LIN {X 0,Y 467.553,Z 325.87,A -85,B 0,C 180,E1 -7518.727,E2 -7518.727} C_VEL
LIN {X 0,Y 467.539,Z 325.868,A -85,B 0,C 180,E1 -7521.952,E2 -7521.952} C_VEL
LIN {X 0,Y 467.553,Z 325.867,A -85,B 0,C 180,E1 -7525.166,E2 -7525.166} C_VEL
LIN {X 0,Y 467.55,Z 325.866,A -85,B 0,C 180,E1 -7528.257,E2 -7528.257} C_VEL
LIN {X 0,Y 467.53,Z 325.867,A -85,B 0,C 180,E1 -7531.247,E2 -7531.247} C_VEL
LIN {X 0,Y 467.581,Z 325.868,A -85,B 0,C 180,E1 -7534.401,E2 -7534.401} C_VEL
LIN {X 0,Y 467.572,Z 325.861,A -85,B 0,C 180,E1 -7536.995,E2 -7536.995} C_VEL
LIN {X 0,Y 467.614,Z 325.847,A -85,B 0,C 180,E1 -7539.776,E2 -7539.776} C_VEL
LIN {X 0,Y 467.566,Z 325.869,A -85,B 0,C 180,E1 -7542.505,E2 -7542.505} C_VEL
LIN {X 0,Y 467.595,Z 325.86,A -85,B 0,C 180,E1 -7545.196,E2 -7545.196} C_VEL
LIN {X 0,Y 467.661,Z 325.849,A -85,B 0,C 180,E1 -7547.854,E2 -7547.854} C_VEL
LIN {X 0,Y 467.67,Z 325.846,A -85,B 0,C 180,E1 -7551.357,E2 -7551.357} C_VEL
LIN {X 0,Y 467.709,Z 325.851,A -85,B 0,C 180,E1 -7553.962,E2 -7553.962} C_VEL
LIN {X 0,Y 467.852,Z 325.827,A -85,B 0,C 180,E1 -7557.417,E2 -7557.417} C_VEL
LIN {X 0,Y 467.853,Z 325.834,A -85,B 0,C 180,E1 -7560,E2 -7560} C_VEL
LIN {X 0,Y 467.818,Z 325.834,A -85,B 0,C 180,E1 -7562.583,E2 -7562.583} C_VEL
LIN {X 0,Y 467.715,Z 325.85,A -85,B 0,C 180,E1 -7566.038,E2 -7566.038} C_VEL
LIN {X 0,Y 467.667,Z 325.852,A -85,B 0,C 180,E1 -7568.643,E2 -7568.643} C_VEL
LIN {X 0,Y 467.66,Z 325.857,A -85,B 0,C 180,E1 -7572.145,E2 -7572.145} C_VEL
LIN {X 0,Y 467.642,Z 325.858,A -85,B 0,C 180,E1 -7575.695,E2 -7575.695} C_VEL
LIN {X 0,Y 467.624,Z 325.857,A -85,B 0,C 180,E1 -7579.308,E2 -7579.308} C_VEL
LIN {X 0,Y 467.538,Z 325.872,A -85,B 0,C 180,E1 -7582.074,E2 -7582.074} C_VEL
LIN {X 0,Y 467.587,Z 325.861,A -85,B 0,C 180,E1 -7584.888,E2 -7584.888} C_VEL
LIN {X 0,Y 467.604,Z 325.867,A -85,B 0,C 180,E1 -7587.77,E2 -7587.77} C_VEL
LIN {X 0,Y 467.571,Z 325.866,A -85,B 0,C 180,E1 -7591.045,E2 -7591.045} C_VEL
LIN {X 0,Y 467.591,Z 325.864,A -85,B 0,C 180,E1 -7594.242,E2 -7594.242} C_VEL
LIN {X 0,Y 467.55,Z 325.87,A -85,B 0,C 180,E1 -7597.186,E2 -7597.186} C_VEL
LIN {X 0,Y 467.579,Z 325.864,A -85,B 0,C 180,E1 -7600.264,E2 -7600.264} C_VEL
LIN {X 0,Y 467.588,Z 325.863,A -85,B 0,C 180,E1 -7602.567,E2 -7602.567} C_VEL
LIN {X 0,Y 467.567,Z 325.867,A -85,B 0,C 180,E1 -7605.052,E2 -7605.052} C_VEL
LIN {X 0,Y 467.59,Z 325.868,A -85,B 0,C 180,E1 -7607.44,E2 -7607.44} C_VEL
LIN {X 0,Y 467.584,Z 325.865,A -85,B 0,C 180,E1 -7610.855,E2 -7610.855} C_VEL
LIN {X 0,Y 467.564,Z 325.869,A -85,B 0,C 180,E1 -7614.26,E2 -7614.26} C_VEL
LIN {X 0,Y 467.583,Z 325.87,A -85,B 0,C 180,E1 -7617.321,E2 -7617.321} C_VEL
LIN {X 0,Y 467.572,Z 325.868,A -85,B 0,C 180,E1 -7620.667,E2 -7620.667} C_VEL
LIN {X 0,Y 467.636,Z 325.967,A -85,B 0,C 180,E1 -7622.232,E2 -7622.232} C_VEL
LIN {X 0,Y 470.731,Z 340.487,A -85,B 0,C 180,E1 -7624.817,E2 -7624.817} C_VEL
LIN {X 0,Y 470.565,Z 347.239,A -85,B 0,C 180,E1 -7625.916,E2 -7625.916} C_VEL
LIN {X 0,Y 469.719,Z 364.781,A -85,B 0,C 180,E1 -7628.726,E2 -7628.726} C_VEL
LIN {X 0,Y 469.507,Z 369.211,A -85,B 0,C 180,E1 -7629.429,E2 -7629.429} C_VEL
LIN {X 0,Y 473.272,Z 391.149,A -85,B 0,C 180,E1 -7629.938,E2 -7629.938} C_VEL
LIN {X 0,Y 472.122,Z 507.018,A -85,B 0,C 180,E1 -7631.727,E2 -7631.727} C_VEL
LIN {X 0,Y 471.734,Z 521.803,A -85,B 0,C 180,E1 -7632.133,E2 -7632.133} C_VEL
LIN {X 0,Y 471.163,Z 535.874,A -85,B 0,C 180,E1 -7632.7,E2 -7632.7} C_VEL
LIN {X 0,Y 470.582,Z 549.218,A -85,B 0,C 180,E1 -7633.423,E2 -7633.423} C_VEL
LIN {X 0,Y 469.899,Z 561.559,A -85,B 0,C 180,E1 -7634.271,E2 -7634.271} C_VEL
LIN {X 0,Y 469.195,Z 573.089,A -85,B 0,C 180,E1 -7635.248,E2 -7635.248} C_VEL
LIN {X 0,Y 468.589,Z 583.675,A -85,B 0,C 180,E1 -7636.336,E2 -7636.336} C_VEL
LIN {X 0,Y 468.153,Z 593.303,A -85,B 0,C 180,E1 -7637.528,E2 -7637.528} C_VEL
LIN {X 0,Y 467.606,Z 602.867,A -85,B 0,C 180,E1 -7638.952,E2 -7638.952} C_VEL
LIN {X 0,Y 467.214,Z 611.173,A -85,B 0,C 180,E1 -7640.476,E2 -7640.476} C_VEL
LIN {X 0,Y 466.951,Z 616.974,A -85,B 0,C 180,E1 -7641.779,E2 -7641.779} C_VEL
LIN {X 0,Y 466.824,Z 621.734,A -85,B 0,C 180,E1 -7643.083,E2 -7643.083} C_VEL
LIN {X 0,Y 466.731,Z 626.661,A -85,B 0,C 180,E1 -7644.816,E2 -7644.816} C_VEL
LIN {X 0,Y 466.679,Z 630.085,A -85,B 0,C 180,E1 -7646.547,E2 -7646.547} C_VEL
LIN {X 0,Y 466.604,Z 632.11,A -85,B 0,C 180,E1 -7648.274,E2 -7648.274} C_VEL
LIN {X 0,Y 466.597,Z 632.785,A -85,B 0,C 180,E1 -7650,E2 -7650} C_VEL
LIN {X 0,Y 466.604,Z 632.119,A -85,B 0,C 180,E1 -7651.726,E2 -7651.726} C_VEL
LIN {X 0,Y 466.679,Z 630.105,A -85,B 0,C 180,E1 -7653.454,E2 -7653.454} C_VEL
LIN {X 0,Y 466.731,Z 626.693,A -85,B 0,C 180,E1 -7655.184,E2 -7655.184} C_VEL
LIN {X 0,Y 466.821,Z 621.783,A -85,B 0,C 180,E1 -7656.918,E2 -7656.918} C_VEL
LIN {X 0,Y 467.036,Z 615.238,A -85,B 0,C 180,E1 -7658.655,E2 -7658.655} C_VEL
LIN {X 0,Y 467.311,Z 607.962,A -85,B 0,C 180,E1 -7660.178,E2 -7660.178} C_VEL
LIN {X 0,Y 467.866,Z 598.973,A -85,B 0,C 180,E1 -7661.7,E2 -7661.7} C_VEL
LIN {X 0,Y 468.352,Z 589.547,A -85,B 0,C 180,E1 -7663.008,E2 -7663.008} C_VEL
LIN {X 0,Y 468.94,Z 579.125,A -85,B 0,C 180,E1 -7664.206,E2 -7664.206} C_VEL
LIN {X 0,Y 469.628,Z 567.65,A -85,B 0,C 180,E1 -7665.293,E2 -7665.293} C_VEL
LIN {X 0,Y 470.388,Z 554.947,A -85,B 0,C 180,E1 -7666.269,E2 -7666.269} C_VEL
LIN {X 0,Y 471.034,Z 542.365,A -85,B 0,C 180,E1 -7667.039,E2 -7667.039} C_VEL
LIN {X 0,Y 471.651,Z 528.534,A -85,B 0,C 180,E1 -7667.691,E2 -7667.691} C_VEL
LIN {X 0,Y 472.117,Z 514.909,A -85,B 0,C 180,E1 -7668.155,E2 -7668.155} C_VEL
LIN {X 0,Y 472.451,Z 501.171,A -85,B 0,C 180,E1 -7668.456,E2 -7668.456} C_VEL
LIN {X 0,Y 473.513,Z 390.833,A -85,B 0,C 180,E1 -7670.162,E2 -7670.162} C_VEL
LIN {X 0,Y 470.004,Z 371.054,A -85,B 0,C 180,E1 -7670.646,E2 -7670.646} C_VEL
LIN {X 0,Y 469.663,Z 369.039,A -85,B 0,C 180,E1 -7670.714,E2 -7670.714} C_VEL
LIN {X 0,Y 470.649,Z 350.152,A -85,B 0,C 180,E1 -7673.777,E2 -7673.777} C_VEL
LIN {X 0,Y 471.053,Z 341.727,A -85,B 0,C 180,E1 -7675.164,E2 -7675.164} C_VEL
LIN {X 0,Y 468.146,Z 328.134,A -85,B 0,C 180,E1 -7677.658,E2 -7677.658} C_VEL
LIN {X 0,Y 467.612,Z 325.864,A -85,B 0,C 180,E1 -7678.135,E2 -7678.135} C_VEL
LIN {X 0,Y 467.584,Z 325.863,A -85,B 0,C 180,E1 -7681.74,E2 -7681.74} C_VEL
LIN {X 0,Y 467.566,Z 325.87,A -85,B 0,C 180,E1 -7684.833,E2 -7684.833} C_VEL
LIN {X 0,Y 467.567,Z 325.868,A -85,B 0,C 180,E1 -7688.045,E2 -7688.045} C_VEL
LIN {X 0,Y 467.58,Z 325.863,A -85,B 0,C 180,E1 -7691.277,E2 -7691.277} C_VEL
LIN {X 0,Y 467.551,Z 325.866,A -85,B 0,C 180,E1 -7693.821,E2 -7693.821} C_VEL
LIN {X 0,Y 467.556,Z 325.869,A -85,B 0,C 180,E1 -7696.256,E2 -7696.256} C_VEL
LIN {X 0,Y 467.58,Z 325.866,A -85,B 0,C 180,E1 -7698.723,E2 -7698.723} C_VEL
LIN {X 0,Y 467.565,Z 325.866,A -85,B 0,C 180,E1 -7701.956,E2 -7701.956} C_VEL
LIN {X 0,Y 467.565,Z 325.865,A -85,B 0,C 180,E1 -7705.168,E2 -7705.168} C_VEL
LIN {X 0,Y 467.586,Z 325.868,A -85,B 0,C 180,E1 -7708.26,E2 -7708.26} C_VEL
LIN {X 0,Y 467.558,Z 325.865,A -85,B 0,C 180,E1 -7711.249,E2 -7711.249} C_VEL
LIN {X 0,Y 467.587,Z 325.864,A -85,B 0,C 180,E1 -7714.159,E2 -7714.159} C_VEL
LIN {X 0,Y 467.579,Z 325.861,A -85,B 0,C 180,E1 -7716.996,E2 -7716.996} C_VEL
LIN {X 0,Y 467.626,Z 325.859,A -85,B 0,C 180,E1 -7719.777,E2 -7719.777} C_VEL
LIN {X 0,Y 467.599,Z 325.861,A -85,B 0,C 180,E1 -7722.507,E2 -7722.507} C_VEL
LIN {X 0,Y 467.609,Z 325.859,A -85,B 0,C 180,E1 -7725.197,E2 -7725.197} C_VEL
LIN {X 0,Y 467.66,Z 325.853,A -85,B 0,C 180,E1 -7727.855,E2 -7727.855} C_VEL
LIN {X 0,Y 467.667,Z 325.85,A -85,B 0,C 180,E1 -7731.357,E2 -7731.357} C_VEL
LIN {X 0,Y 467.715,Z 325.853,A -85,B 0,C 180,E1 -7733.962,E2 -7733.962} C_VEL
LIN {X 0,Y 467.818,Z 325.829,A -85,B 0,C 180,E1 -7737.417,E2 -7737.417} C_VEL
LIN {X 0,Y 467.853,Z 325.833,A -85,B 0,C 180,E1 -7740,E2 -7740} C_VEL
LIN {X 0,Y 467.852,Z 325.827,A -85,B 0,C 180,E1 -7742.583,E2 -7742.583} C_VEL
LIN {X 0,Y 467.705,Z 325.846,A -85,B 0,C 180,E1 -7746.038,E2 -7746.038} C_VEL
LIN {X 0,Y 467.662,Z 325.852,A -85,B 0,C 180,E1 -7748.643,E2 -7748.643} C_VEL
LIN {X 0,Y 467.661,Z 325.853,A -85,B 0,C 180,E1 -7752.146,E2 -7752.146} C_VEL
LIN {X 0,Y 467.616,Z 325.86,A -85,B 0,C 180,E1 -7755.696,E2 -7755.696} C_VEL
LIN {X 0,Y 467.581,Z 325.862,A -85,B 0,C 180,E1 -7758.75,E2 -7758.75} C_VEL
LIN {X 0,Y 467.562,Z 325.864,A -85,B 0,C 180,E1 -7761.261,E2 -7761.261} C_VEL
LIN {X 0,Y 467.558,Z 325.865,A -85,B 0,C 180,E1 -7763.944,E2 -7763.944} C_VEL
LIN {X 0,Y 467.538,Z 325.868,A -85,B 0,C 180,E1 -7766.806,E2 -7766.806} C_VEL
LIN {X 0,Y 467.513,Z 325.861,A -85,B 0,C 180,E1 -7769.741,E2 -7769.741} C_VEL
LIN {X 0,Y 467.574,Z 325.862,A -85,B 0,C 180,E1 -7772.76,E2 -7772.76} C_VEL
LIN {X 0,Y 467.545,Z 325.859,A -85,B 0,C 180,E1 -7775.891,E2 -7775.891} C_VEL
LIN {X 0,Y 467.531,Z 325.873,A -85,B 0,C 180,E1 -7779.15,E2 -7779.15} C_VEL
LIN {X 0,Y 467.553,Z 325.873,A -85,B 0,C 180,E1 -7781.406,E2 -7781.406} C_VEL
LIN {X 0,Y 467.565,Z 325.869,A -85,B 0,C 180,E1 -7785.052,E2 -7785.052} C_VEL
LIN {X 0,Y 467.553,Z 325.87,A -85,B 0,C 180,E1 -7788.727,E2 -7788.727} C_VEL
LIN {X 0,Y 467.536,Z 325.872,A -85,B 0,C 180,E1 -7791.952,E2 -7791.952} C_VEL
LIN {X 0,Y 467.544,Z 325.874,A -85,B 0,C 180,E1 -7795.165,E2 -7795.165} C_VEL
LIN {X 0,Y 467.546,Z 325.868,A -85,B 0,C 180,E1 -7798.257,E2 -7798.257} C_VEL
LIN {X 0,Y 467.574,Z 326.065,A -85,B 0,C 180,E1 -7800.51,E2 -7800.51} C_VEL
LIN {X 0,Y 469.898,Z 337.319,A -85,B 0,C 180,E1 -7802.859,E2 -7802.859} C_VEL
LIN {X 0,Y 469.985,Z 342.162,A -85,B 0,C 180,E1 -7803.796,E2 -7803.796} C_VEL
LIN {X 0,Y 469.828,Z 345.296,A -85,B 0,C 180,E1 -7804.37,E2 -7804.37} C_VEL
LIN {X 0,Y 473.739,Z 362.985,A -85,B 0,C 180,E1 -7804.845,E2 -7804.845} C_VEL
LIN {X 0,Y 473.314,Z 405.55,A -85,B 0,C 180,E1 -7805.504,E2 -7805.504} C_VEL
LIN {X 0,Y 472.705,Z 411.397,A -85,B 0,C 180,E1 -7805.569,E2 -7805.569} C_VEL
LIN {X 0,Y 467.064,Z 430.434,A -85,B 0,C 180,E1 -7805.612,E2 -7805.612} C_VEL
LIN {X 0,Y 466.356,Z 436.288,A -85,B 0,C 180,E1 -7805.674,E2 -7805.674} C_VEL
LIN {X 0,Y 465.947,Z 481.822,A -85,B 0,C 180,E1 -7806.411,E2 -7806.411} C_VEL
LIN {X 0,Y 465.524,Z 495.912,A -85,B 0,C 180,E1 -7806.8,E2 -7806.8} C_VEL
LIN {X 0,Y 464.986,Z 508.239,A -85,B 0,C 180,E1 -7807.288,E2 -7807.288} C_VEL
LIN {X 0,Y 464.373,Z 521.643,A -85,B 0,C 180,E1 -7808.002,E2 -7808.002} C_VEL
LIN {X 0,Y 463.638,Z 534.729,A -85,B 0,C 180,E1 -7808.899,E2 -7808.899} C_VEL
LIN {X 0,Y 462.972,Z 545.605,A -85,B 0,C 180,E1 -7809.82,E2 -7809.82} C_VEL
LIN {X 0,Y 462.286,Z 556.356,A -85,B 0,C 180,E1 -7810.922,E2 -7810.922} C_VEL
LIN {X 0,Y 461.558,Z 567.169,A -85,B 0,C 180,E1 -7812.27,E2 -7812.27} C_VEL
LIN {X 0,Y 461.008,Z 576.208,A -85,B 0,C 180,E1 -7813.643,E2 -7813.643} C_VEL
LIN {X 0,Y 460.571,Z 583.422,A -85,B 0,C 180,E1 -7814.965,E2 -7814.965} C_VEL
LIN {X 0,Y 460.181,Z 589.526,A -85,B 0,C 180,E1 -7816.307,E2 -7816.307} C_VEL
LIN {X 0,Y 459.834,Z 595.712,A -85,B 0,C 180,E1 -7818.006,E2 -7818.006} C_VEL
LIN {X 0,Y 459.725,Z 599.724,A -85,B 0,C 180,E1 -7819.429,E2 -7819.429} C_VEL
LIN {X 0,Y 459.57,Z 603.358,A -85,B 0,C 180,E1 -7821.203,E2 -7821.203} C_VEL
LIN {X 0,Y 459.576,Z 605.577,A -85,B 0,C 180,E1 -7822.973,E2 -7822.973} C_VEL
LIN {X 0,Y 459.558,Z 606.452,A -85,B 0,C 180,E1 -7824.735,E2 -7824.735} C_VEL
LIN {X 0,Y 459.563,Z 606.007,A -85,B 0,C 180,E1 -7826.493,E2 -7826.493} C_VEL
LIN {X 0,Y 459.572,Z 604.245,A -85,B 0,C 180,E1 -7828.247,E2 -7828.247} C_VEL
LIN {X 0,Y 459.571,Z 601.136,A -85,B 0,C 180,E1 -7830,E2 -7830} C_VEL
LIN {X 0,Y 459.707,Z 596.563,A -85,B 0,C 180,E1 -7831.752,E2 -7831.752} C_VEL
LIN {X 0,Y 460.099,Z 590.362,A -85,B 0,C 180,E1 -7833.503,E2 -7833.503} C_VEL
LIN {X 0,Y 460.54,Z 583.469,A -85,B 0,C 180,E1 -7835.034,E2 -7835.034} C_VEL
LIN {X 0,Y 461.001,Z 574.951,A -85,B 0,C 180,E1 -7836.565,E2 -7836.565} C_VEL
LIN {X 0,Y 461.415,Z 567.702,A -85,B 0,C 180,E1 -7837.654,E2 -7837.654} C_VEL
LIN {X 0,Y 461.983,Z 559.151,A -85,B 0,C 180,E1 -7838.75,E2 -7838.75} C_VEL
LIN {X 0,Y 462.709,Z 547.862,A -85,B 0,C 180,E1 -7839.949,E2 -7839.949} C_VEL
LIN {X 0,Y 463.353,Z 536.647,A -85,B 0,C 180,E1 -7840.929,E2 -7840.929} C_VEL
LIN {X 0,Y 464.007,Z 524.401,A -85,B 0,C 180,E1 -7841.799,E2 -7841.799} C_VEL
LIN {X 0,Y 464.565,Z 510.773,A -85,B 0,C 180,E1 -7842.56,E2 -7842.56} C_VEL
LIN {X 0,Y 465.159,Z 497.073,A -85,B 0,C 180,E1 -7843.127,E2 -7843.127} C_VEL
LIN {X 0,Y 465.47,Z 482.92,A -85,B 0,C 180,E1 -7843.535,E2 -7843.535} C_VEL
LIN {X 0,Y 465.999,Z 437.32,A -85,B 0,C 180,E1 -7844.269,E2 -7844.269} C_VEL
LIN {X 0,Y 466.607,Z 363.158,A -85,B 0,C 180,E1 -7845.427,E2 -7845.427} C_VEL
LIN {X 0,Y 462.751,Z 345.257,A -85,B 0,C 180,E1 -7845.893,E2 -7845.893} C_VEL
LIN {X 0,Y 462.849,Z 338.115,A -85,B 0,C 180,E1 -7847.252,E2 -7847.252} C_VEL
LIN {X 0,Y 460.57,Z 326.743,A -85,B 0,C 180,E1 -7849.616,E2 -7849.616} C_VEL
LIN {X 0,Y 460.499,Z 326.75,A -85,B 0,C 180,E1 -7852.429,E2 -7852.429} C_VEL
LIN {X 0,Y 460.524,Z 326.745,A -85,B 0,C 180,E1 -7855.789,E2 -7855.789} C_VEL
LIN {X 0,Y 460.499,Z 326.748,A -85,B 0,C 180,E1 -7858.237,E2 -7858.237} C_VEL
LIN {X 0,Y 460.499,Z 326.748,A -85,B 0,C 180,E1 -7861.277,E2 -7861.277} C_VEL
LIN {X 0,Y 460.512,Z 326.748,A -85,B 0,C 180,E1 -7864.501,E2 -7864.501} C_VEL
LIN {X 0,Y 460.481,Z 326.747,A -85,B 0,C 180,E1 -7867.625,E2 -7867.625} C_VEL
LIN {X 0,Y 460.502,Z 326.747,A -85,B 0,C 180,E1 -7871.015,E2 -7871.015} C_VEL
LIN {X 0,Y 460.513,Z 326.748,A -85,B 0,C 180,E1 -7874.589,E2 -7874.589} C_VEL
LIN {X 0,Y 460.473,Z 326.747,A -85,B 0,C 180,E1 -7877.812,E2 -7877.812} C_VEL
LIN {X 0,Y 460.477,Z 326.749,A -85,B 0,C 180,E1 -7880.131,E2 -7880.131} C_VEL
LIN {X 0,Y 460.461,Z 326.747,A -85,B 0,C 180,E1 -7883.469,E2 -7883.469} C_VEL
LIN {X 0,Y 460.518,Z 326.743,A -85,B 0,C 180,E1 -7886.674,E2 -7886.674} C_VEL
LIN {X 0,Y 460.482,Z 326.747,A -85,B 0,C 180,E1 -7889.757,E2 -7889.757} C_VEL
LIN {X 0,Y 460.493,Z 326.746,A -85,B 0,C 180,E1 -7892.751,E2 -7892.751} C_VEL
LIN {X 0,Y 460.52,Z 326.742,A -85,B 0,C 180,E1 -7895.666,E2 -7895.666} C_VEL
LIN {X 0,Y 460.522,Z 326.734,A -85,B 0,C 180,E1 -7898.579,E2 -7898.579} C_VEL
LIN {X 0,Y 460.585,Z 326.727,A -85,B 0,C 180,E1 -7901.31,E2 -7901.31} C_VEL
LIN {X 0,Y 460.552,Z 326.738,A -85,B 0,C 180,E1 -7904.964,E2 -7904.964} C_VEL
LIN {X 0,Y 460.613,Z 326.717,A -85,B 0,C 180,E1 -7908.559,E2 -7908.559} C_VEL
LIN {X 0,Y 460.621,Z 326.724,A -85,B 0,C 180,E1 -7911.223,E2 -7911.223} C_VEL
LIN {X 0,Y 460.675,Z 326.726,A -85,B 0,C 180,E1 -7913.869,E2 -7913.869} C_VEL
LIN {X 0,Y 460.792,Z 326.707,A -85,B 0,C 180,E1 -7917.377,E2 -7917.377} C_VEL
LIN {X 0,Y 460.823,Z 326.71,A -85,B 0,C 180,E1 -7920,E2 -7920} C_VEL
LIN {X 0,Y 460.762,Z 326.713,A -85,B 0,C 180,E1 -7922.622,E2 -7922.622} C_VEL
LIN {X 0,Y 460.679,Z 326.727,A -85,B 0,C 180,E1 -7926.13,E2 -7926.13} C_VEL
LIN {X 0,Y 460.618,Z 326.729,A -85,B 0,C 180,E1 -7928.776,E2 -7928.776} C_VEL
LIN {X 0,Y 460.617,Z 326.731,A -85,B 0,C 180,E1 -7932.445,E2 -7932.445} C_VEL
LIN {X 0,Y 460.604,Z 326.738,A -85,B 0,C 180,E1 -7935.997,E2 -7935.997} C_VEL
LIN {X 0,Y 460.571,Z 326.739,A -85,B 0,C 180,E1 -7939.615,E2 -7939.615} C_VEL
LIN {X 0,Y 460.514,Z 326.743,A -85,B 0,C 180,E1 -7942.428,E2 -7942.428} C_VEL
LIN {X 0,Y 460.548,Z 326.744,A -85,B 0,C 180,E1 -7945.796,E2 -7945.796} C_VEL
LIN {X 0,Y 460.538,Z 326.741,A -85,B 0,C 180,E1 -7948.234,E2 -7948.234} C_VEL
LIN {X 0,Y 460.523,Z 326.746,A -85,B 0,C 180,E1 -7951.283,E2 -7951.283} C_VEL
LIN {X 0,Y 460.534,Z 326.742,A -85,B 0,C 180,E1 -7954.505,E2 -7954.505} C_VEL
LIN {X 0,Y 460.529,Z 326.749,A -85,B 0,C 180,E1 -7957.62,E2 -7957.62} C_VEL
LIN {X 0,Y 460.544,Z 326.741,A -85,B 0,C 180,E1 -7960.269,E2 -7960.269} C_VEL
LIN {X 0,Y 460.501,Z 326.751,A -85,B 0,C 180,E1 -7963.375,E2 -7963.375} C_VEL
LIN {X 0,Y 460.5,Z 326.745,A -85,B 0,C 180,E1 -7966.624,E2 -7966.624} C_VEL
LIN {X 0,Y 460.543,Z 326.745,A -85,B 0,C 180,E1 -7969.73,E2 -7969.73} C_VEL
LIN {X 0,Y 460.528,Z 326.745,A -85,B 0,C 180,E1 -7972.519,E2 -7972.519} C_VEL
LIN {X 0,Y 460.55,Z 326.746,A -85,B 0,C 180,E1 -7975.624,E2 -7975.624} C_VEL
LIN {X 0,Y 460.538,Z 326.743,A -85,B 0,C 180,E1 -7978.744,E2 -7978.744} C_VEL
LIN {X 0,Y 460.593,Z 326.831,A -85,B 0,C 180,E1 -7981.979,E2 -7981.979} C_VEL
LIN {X 0,Y 463.754,Z 341.584,A -85,B 0,C 180,E1 -7984.652,E2 -7984.652} C_VEL
LIN {X 0,Y 463.763,Z 346.87,A -85,B 0,C 180,E1 -7985.533,E2 -7985.533} C_VEL
LIN {X 0,Y 462.75,Z 365.877,A -85,B 0,C 180,E1 -7988.623,E2 -7988.623} C_VEL
LIN {X 0,Y 462.598,Z 369.02,A -85,B 0,C 180,E1 -7989.131,E2 -7989.131} C_VEL
LIN {X 0,Y 466.544,Z 392.063,A -85,B 0,C 180,E1 -7989.673,E2 -7989.673} C_VEL
LIN {X 0,Y 465.333,Z 507.257,A -85,B 0,C 180,E1 -7991.48,E2 -7991.48} C_VEL
LIN {X 0,Y 464.919,Z 521.888,A -85,B 0,C 180,E1 -7991.89,E2 -7991.89} C_VEL
LIN {X 0,Y 464.342,Z 535.865,A -85,B 0,C 180,E1 -7992.464,E2 -7992.464} C_VEL
LIN {X 0,Y 463.733,Z 548.889,A -85,B 0,C 180,E1 -7993.18,E2 -7993.18} C_VEL
LIN {X 0,Y 463.03,Z 561.144,A -85,B 0,C 180,E1 -7994.032,E2 -7994.032} C_VEL
LIN {X 0,Y 462.289,Z 572.719,A -85,B 0,C 180,E1 -7995.022,E2 -7995.022} C_VEL
LIN {X 0,Y 461.632,Z 583.336,A -85,B 0,C 180,E1 -7996.126,E2 -7996.126} C_VEL
LIN {X 0,Y 461.123,Z 593.72,A -85,B 0,C 180,E1 -7997.434,E2 -7997.434} C_VEL
LIN {X 0,Y 460.601,Z 602.579,A -85,B 0,C 180,E1 -7998.782,E2 -7998.782} C_VEL
LIN {X 0,Y 460.142,Z 610.908,A -85,B 0,C 180,E1 -8000.328,E2 -8000.328} C_VEL
LIN {X 0,Y 459.896,Z 616.719,A -85,B 0,C 180,E1 -8001.652,E2 -8001.652} C_VEL
LIN {X 0,Y 459.733,Z 621.492,A -85,B 0,C 180,E1 -8002.975,E2 -8002.975} C_VEL
LIN {X 0,Y 459.644,Z 626.432,A -85,B 0,C 180,E1 -8004.736,E2 -8004.736} C_VEL
LIN {X 0,Y 459.574,Z 629.866,A -85,B 0,C 180,E1 -8006.493,E2 -8006.493} C_VEL
LIN {X 0,Y 459.517,Z 631.9,A -85,B 0,C 180,E1 -8008.247,E2 -8008.247} C_VEL
LIN {X 0,Y 459.528,Z 632.584,A -85,B 0,C 180,E1 -8010,E2 -8010} C_VEL
LIN {X 0,Y 459.517,Z 631.926,A -85,B 0,C 180,E1 -8011.753,E2 -8011.753} C_VEL
LIN {X 0,Y 459.574,Z 629.92,A -85,B 0,C 180,E1 -8013.507,E2 -8013.507} C_VEL
LIN {X 0,Y 459.645,Z 626.518,A -85,B 0,C 180,E1 -8015.264,E2 -8015.264} C_VEL
LIN {X 0,Y 459.731,Z 621.621,A -85,B 0,C 180,E1 -8017.025,E2 -8017.025} C_VEL
LIN {X 0,Y 459.969,Z 615.089,A -85,B 0,C 180,E1 -8018.789,E2 -8018.789} C_VEL
LIN {X 0,Y 460.28,Z 607.829,A -85,B 0,C 180,E1 -8020.336,E2 -8020.336} C_VEL
LIN {X 0,Y 460.856,Z 598.866,A -85,B 0,C 180,E1 -8021.881,E2 -8021.881} C_VEL
LIN {X 0,Y 461.374,Z 589.468,A -85,B 0,C 180,E1 -8023.208,E2 -8023.208} C_VEL
LIN {X 0,Y 462.008,Z 579.079,A -85,B 0,C 180,E1 -8024.424,E2 -8024.424} C_VEL
LIN {X 0,Y 462.766,Z 567.642,A -85,B 0,C 180,E1 -8025.526,E2 -8025.526} C_VEL
LIN {X 0,Y 463.561,Z 554.989,A -85,B 0,C 180,E1 -8026.515,E2 -8026.515} C_VEL
LIN {X 0,Y 464.308,Z 541.922,A -85,B 0,C 180,E1 -8027.326,E2 -8027.326} C_VEL
LIN {X 0,Y 464.905,Z 527.983,A -85,B 0,C 180,E1 -8027.99,E2 -8027.99} C_VEL
LIN {X 0,Y 465.475,Z 513.268,A -85,B 0,C 180,E1 -8028.486,E2 -8028.486} C_VEL
LIN {X 0,Y 465.787,Z 498.747,A -85,B 0,C 180,E1 -8028.787,E2 -8028.787} C_VEL
LIN {X 0,Y 466.906,Z 391.754,A -85,B 0,C 180,E1 -8030.462,E2 -8030.462} C_VEL
LIN {X 0,Y 463.435,Z 372.229,A -85,B 0,C 180,E1 -8030.951,E2 -8030.951} C_VEL
LIN {X 0,Y 462.798,Z 368.937,A -85,B 0,C 180,E1 -8031.04,E2 -8031.04} C_VEL
LIN {X 0,Y 463.768,Z 351.507,A -85,B 0,C 180,E1 -8033.915,E2 -8033.915} C_VEL
LIN {X 0,Y 464.155,Z 343.091,A -85,B 0,C 180,E1 -8035.325,E2 -8035.325} C_VEL
LIN {X 0,Y 461.437,Z 330.397,A -85,B 0,C 180,E1 -8037.694,E2 -8037.694} C_VEL
LIN {X 0,Y 460.575,Z 326.74,A -85,B 0,C 180,E1 -8038.418,E2 -8038.418} C_VEL
LIN {X 0,Y 460.523,Z 326.744,A -85,B 0,C 180,E1 -8041.283,E2 -8041.283} C_VEL
LIN {X 0,Y 460.533,Z 326.747,A -85,B 0,C 180,E1 -8044.506,E2 -8044.506} C_VEL
LIN {X 0,Y 460.503,Z 326.746,A -85,B 0,C 180,E1 -8047.623,E2 -8047.623} C_VEL
LIN {X 0,Y 460.541,Z 326.744,A -85,B 0,C 180,E1 -8050.269,E2 -8050.269} C_VEL
LIN {X 0,Y 460.498,Z 326.743,A -85,B 0,C 180,E1 -8053.376,E2 -8053.376} C_VEL
LIN {X 0,Y 460.501,Z 326.75,A -85,B 0,C 180,E1 -8056.625,E2 -8056.625} C_VEL
LIN {X 0,Y 460.544,Z 326.74,A -85,B 0,C 180,E1 -8059.731,E2 -8059.731} C_VEL
LIN {X 0,Y 460.499,Z 326.748,A -85,B 0,C 180,E1 -8062.525,E2 -8062.525} C_VEL
LIN {X 0,Y 460.548,Z 326.739,A -85,B 0,C 180,E1 -8065.624,E2 -8065.624} C_VEL
LIN {X 0,Y 460.54,Z 326.741,A -85,B 0,C 180,E1 -8068.745,E2 -8068.745} C_VEL
LIN {X 0,Y 460.553,Z 326.744,A -85,B 0,C 180,E1 -8072.262,E2 -8072.262} C_VEL
LIN {X 0,Y 460.543,Z 326.741,A -85,B 0,C 180,E1 -8074.705,E2 -8074.705} C_VEL
LIN {X 0,Y 460.514,Z 326.742,A -85,B 0,C 180,E1 -8077.572,E2 -8077.572} C_VEL
LIN {X 0,Y 460.571,Z 326.739,A -85,B 0,C 180,E1 -8080.385,E2 -8080.385} C_VEL
LIN {X 0,Y 460.608,Z 326.737,A -85,B 0,C 180,E1 -8084.059,E2 -8084.059} C_VEL
LIN {X 0,Y 460.613,Z 326.728,A -85,B 0,C 180,E1 -8087.666,E2 -8087.666} C_VEL
LIN {X 0,Y 460.619,Z 326.727,A -85,B 0,C 180,E1 -8091.224,E2 -8091.224} C_VEL
LIN {X 0,Y 460.679,Z 326.727,A -85,B 0,C 180,E1 -8093.87,E2 -8093.87} C_VEL
LIN {X 0,Y 460.762,Z 326.708,A -85,B 0,C 180,E1 -8097.378,E2 -8097.378} C_VEL
LIN {X 0,Y 460.823,Z 326.708,A -85,B 0,C 180,E1 -8100,E2 -8100} C_VEL
LIN {X 0,Y 460.792,Z 326.706,A -85,B 0,C 180,E1 -8102.623,E2 -8102.623} C_VEL
LIN {X 0,Y 460.671,Z 326.721,A -85,B 0,C 180,E1 -8106.131,E2 -8106.131} C_VEL
LIN {X 0,Y 460.614,Z 326.73,A -85,B 0,C 180,E1 -8108.777,E2 -8108.777} C_VEL
LIN {X 0,Y 460.614,Z 326.729,A -85,B 0,C 180,E1 -8112.334,E2 -8112.334} C_VEL
LIN {X 0,Y 460.561,Z 326.736,A -85,B 0,C 180,E1 -8115.978,E2 -8115.978} C_VEL
LIN {X 0,Y 460.539,Z 326.74,A -85,B 0,C 180,E1 -8118.888,E2 -8118.888} C_VEL
LIN {X 0,Y 460.513,Z 326.744,A -85,B 0,C 180,E1 -8121.486,E2 -8121.486} C_VEL
LIN {X 0,Y 460.521,Z 326.739,A -85,B 0,C 180,E1 -8124.334,E2 -8124.334} C_VEL
LIN {X 0,Y 460.493,Z 326.75,A -85,B 0,C 180,E1 -8127.249,E2 -8127.249} C_VEL
LIN {X 0,Y 460.481,Z 326.733,A -85,B 0,C 180,E1 -8130.243,E2 -8130.243} C_VEL
LIN {X 0,Y 460.519,Z 326.747,A -85,B 0,C 180,E1 -8133.326,E2 -8133.326} C_VEL
LIN {X 0,Y 460.46,Z 326.738,A -85,B 0,C 180,E1 -8136.531,E2 -8136.531} C_VEL
LIN {X 0,Y 460.477,Z 326.748,A -85,B 0,C 180,E1 -8139.869,E2 -8139.869} C_VEL
LIN {X 0,Y 460.46,Z 326.752,A -85,B 0,C 180,E1 -8142.893,E2 -8142.893} C_VEL
LIN {X 0,Y 460.507,Z 326.743,A -85,B 0,C 180,E1 -8145.832,E2 -8145.832} C_VEL
LIN {X 0,Y 460.502,Z 326.748,A -85,B 0,C 180,E1 -8148.985,E2 -8148.985} C_VEL
LIN {X 0,Y 460.481,Z 326.75,A -85,B 0,C 180,E1 -8152.375,E2 -8152.375} C_VEL
LIN {X 0,Y 460.526,Z 326.745,A -85,B 0,C 180,E1 -8155.622,E2 -8155.622} C_VEL
LIN {X 0,Y 460.508,Z 326.748,A -85,B 0,C 180,E1 -8158.742,E2 -8158.742} C_VEL
LIN {X 0,Y 460.489,Z 326.821,A -85,B 0,C 180,E1 -8160.194,E2 -8160.194} C_VEL
LIN {X 0,Y 462.943,Z 338.423,A -85,B 0,C 180,E1 -8162.662,E2 -8162.662} C_VEL
LIN {X 0,Y 463.135,Z 342.907,A -85,B 0,C 180,E1 -8163.55,E2 -8163.55} C_VEL
LIN {X 0,Y 463.039,Z 345.659,A -85,B 0,C 180,E1 -8164.033,E2 -8164.033} C_VEL
LIN {X 0,Y 467.072,Z 363.728,A -85,B 0,C 180,E1 -8164.532,E2 -8164.532} C_VEL
LIN {X 0,Y 466.356,Z 436.288,A -85,B 0,C 180,E1 -8165.674,E2 -8165.674} C_VEL
LIN {X 0,Y 465.687,Z 442.128,A -85,B 0,C 180,E1 -8165.737,E2 -8165.737} C_VEL
LIN {X 0,Y 460.198,Z 461.163,A -85,B 0,C 180,E1 -8165.788,E2 -8165.788} C_VEL
LIN {X 0,Y 459.468,Z 467.007,A -85,B 0,C 180,E1 -8165.849,E2 -8165.849} C_VEL
LIN {X 0,Y 459.186,Z 485.434,A -85,B 0,C 180,E1 -8166.191,E2 -8166.191} C_VEL
LIN {X 0,Y 458.667,Z 499.82,A -85,B 0,C 180,E1 -8166.638,E2 -8166.638} C_VEL
LIN {X 0,Y 458.115,Z 513.131,A -85,B 0,C 180,E1 -8167.233,E2 -8167.233} C_VEL
LIN {X 0,Y 457.405,Z 526.288,A -85,B 0,C 180,E1 -8168.005,E2 -8168.005} C_VEL
LIN {X 0,Y 456.64,Z 538.493,A -85,B 0,C 180,E1 -8168.915,E2 -8168.915} C_VEL
LIN {X 0,Y 455.901,Z 549.895,A -85,B 0,C 180,E1 -8169.964,E2 -8169.964} C_VEL
LIN {X 0,Y 455.165,Z 559.958,A -85,B 0,C 180,E1 -8171.08,E2 -8171.08} C_VEL
LIN {X 0,Y 454.435,Z 570.128,A -85,B 0,C 180,E1 -8172.448,E2 -8172.448} C_VEL
LIN {X 0,Y 453.902,Z 578.54,A -85,B 0,C 180,E1 -8173.817,E2 -8173.817} C_VEL
LIN {X 0,Y 453.346,Z 586.545,A -85,B 0,C 180,E1 -8175.409,E2 -8175.409} C_VEL
LIN {X 0,Y 452.989,Z 592.958,A -85,B 0,C 180,E1 -8176.999,E2 -8176.999} C_VEL
LIN {X 0,Y 452.69,Z 598.617,A -85,B 0,C 180,E1 -8178.81,E2 -8178.81} C_VEL
LIN {X 0,Y 452.524,Z 601.803,A -85,B 0,C 180,E1 -8180.163,E2 -8180.163} C_VEL
LIN {X 0,Y 452.477,Z 604.763,A -85,B 0,C 180,E1 -8181.964,E2 -8181.964} C_VEL
LIN {X 0,Y 452.518,Z 606.347,A -85,B 0,C 180,E1 -8183.759,E2 -8183.759} C_VEL
LIN {X 0,Y 452.435,Z 606.607,A -85,B 0,C 180,E1 -8185.545,E2 -8185.545} C_VEL
LIN {X 0,Y 452.516,Z 605.547,A -85,B 0,C 180,E1 -8187.329,E2 -8187.329} C_VEL
LIN {X 0,Y 452.466,Z 603.165,A -85,B 0,C 180,E1 -8189.11,E2 -8189.11} C_VEL
LIN {X 0,Y 452.55,Z 599.399,A -85,B 0,C 180,E1 -8190.89,E2 -8190.89} C_VEL
LIN {X 0,Y 452.83,Z 594.093,A -85,B 0,C 180,E1 -8192.669,E2 -8192.669} C_VEL
LIN {X 0,Y 453.226,Z 589.013,A -85,B 0,C 180,E1 -8194.001,E2 -8194.001} C_VEL
LIN {X 0,Y 453.644,Z 581.763,A -85,B 0,C 180,E1 -8195.556,E2 -8195.556} C_VEL
LIN {X 0,Y 454.202,Z 572.769,A -85,B 0,C 180,E1 -8197.111,E2 -8197.111} C_VEL
LIN {X 0,Y 454.591,Z 564.937,A -85,B 0,C 180,E1 -8198.243,E2 -8198.243} C_VEL
LIN {X 0,Y 455.428,Z 554.025,A -85,B 0,C 180,E1 -8199.549,E2 -8199.549} C_VEL
LIN {X 0,Y 456.101,Z 542.773,A -85,B 0,C 180,E1 -8200.656,E2 -8200.656} C_VEL
LIN {X 0,Y 456.838,Z 530.327,A -85,B 0,C 180,E1 -8201.649,E2 -8201.649} C_VEL
LIN {X 0,Y 457.482,Z 518.286,A -85,B 0,C 180,E1 -8202.42,E2 -8202.42} C_VEL
LIN {X 0,Y 458.086,Z 506.307,A -85,B 0,C 180,E1 -8203.023,E2 -8203.023} C_VEL
LIN {X 0,Y 458.513,Z 492.369,A -85,B 0,C 180,E1 -8203.546,E2 -8203.546} C_VEL
LIN {X 0,Y 458.789,Z 479.205,A -85,B 0,C 180,E1 -8203.877,E2 -8203.877} C_VEL
LIN {X 0,Y 459.926,Z 364.299,A -85,B 0,C 180,E1 -8205.699,E2 -8205.699} C_VEL
LIN {X 0,Y 455.878,Z 345.462,A -85,B 0,C 180,E1 -8206.197,E2 -8206.197} C_VEL
LIN {X 0,Y 456.044,Z 340.44,A -85,B 0,C 180,E1 -8207.161,E2 -8207.161} C_VEL
LIN {X 0,Y 453.511,Z 327.622,A -85,B 0,C 180,E1 -8209.854,E2 -8209.854} C_VEL
LIN {X 0,Y 453.467,Z 327.628,A -85,B 0,C 180,E1 -8212.797,E2 -8212.797} C_VEL
LIN {X 0,Y 453.469,Z 327.624,A -85,B 0,C 180,E1 -8215.985,E2 -8215.985} C_VEL
LIN {X 0,Y 453.451,Z 327.63,A -85,B 0,C 180,E1 -8218.716,E2 -8218.716} C_VEL
LIN {X 0,Y 453.437,Z 327.625,A -85,B 0,C 180,E1 -8221.802,E2 -8221.802} C_VEL
LIN {X 0,Y 453.469,Z 327.626,A -85,B 0,C 180,E1 -8224.99,E2 -8224.99} C_VEL
LIN {X 0,Y 453.44,Z 327.627,A -85,B 0,C 180,E1 -8228.314,E2 -8228.314} C_VEL
LIN {X 0,Y 453.467,Z 327.627,A -85,B 0,C 180,E1 -8230.612,E2 -8230.612} C_VEL
LIN {X 0,Y 453.483,Z 327.624,A -85,B 0,C 180,E1 -8234.528,E2 -8234.528} C_VEL
LIN {X 0,Y 453.433,Z 327.626,A -85,B 0,C 180,E1 -8238.072,E2 -8238.072} C_VEL
LIN {X 0,Y 453.426,Z 327.63,A -85,B 0,C 180,E1 -8240.804,E2 -8240.804} C_VEL
LIN {X 0,Y 453.444,Z 327.623,A -85,B 0,C 180,E1 -8243.916,E2 -8243.916} C_VEL
LIN {X 0,Y 453.483,Z 327.617,A -85,B 0,C 180,E1 -8246.813,E2 -8246.813} C_VEL
LIN {X 0,Y 453.45,Z 327.628,A -85,B 0,C 180,E1 -8250.266,E2 -8250.266} C_VEL
LIN {X 0,Y 453.444,Z 327.62,A -85,B 0,C 180,E1 -8253.29,E2 -8253.29} C_VEL
LIN {X 0,Y 453.495,Z 327.623,A -85,B 0,C 180,E1 -8256.238,E2 -8256.238} C_VEL
LIN {X 0,Y 453.477,Z 327.606,A -85,B 0,C 180,E1 -8259.117,E2 -8259.117} C_VEL
LIN {X 0,Y 453.487,Z 327.614,A -85,B 0,C 180,E1 -8261.943,E2 -8261.943} C_VEL
LIN {X 0,Y 453.522,Z 327.615,A -85,B 0,C 180,E1 -8264.725,E2 -8264.725} C_VEL
LIN {X 0,Y 453.562,Z 327.596,A -85,B 0,C 180,E1 -8268.379,E2 -8268.379} C_VEL
LIN {X 0,Y 453.587,Z 327.6,A -85,B 0,C 180,E1 -8271.086,E2 -8271.086} C_VEL
LIN {X 0,Y 453.642,Z 327.601,A -85,B 0,C 180,E1 -8273.774,E2 -8273.774} C_VEL
LIN {X 0,Y 453.736,Z 327.585,A -85,B 0,C 180,E1 -8277.336,E2 -8277.336} C_VEL
LIN {X 0,Y 453.792,Z 327.585,A -85,B 0,C 180,E1 -8280,E2 -8280} C_VEL
LIN {X 0,Y 453.709,Z 327.591,A -85,B 0,C 180,E1 -8282.663,E2 -8282.663} C_VEL
LIN {X 0,Y 453.646,Z 327.603,A -85,B 0,C 180,E1 -8286.226,E2 -8286.226} C_VEL
LIN {X 0,Y 453.585,Z 327.605,A -85,B 0,C 180,E1 -8288.913,E2 -8288.913} C_VEL
LIN {X 0,Y 453.567,Z 327.609,A -85,B 0,C 180,E1 -8292.529,E2 -8292.529} C_VEL
LIN {X 0,Y 453.547,Z 327.614,A -85,B 0,C 180,E1 -8296.196,E2 -8296.196} C_VEL
LIN {X 0,Y 453.519,Z 327.612,A -85,B 0,C 180,E1 -8299.039,E2 -8299.039} C_VEL
LIN {X 0,Y 453.479,Z 327.623,A -85,B 0,C 180,E1 -8301.836,E2 -8301.836} C_VEL
LIN {X 0,Y 453.502,Z 327.616,A -85,B 0,C 180,E1 -8304.735,E2 -8304.735} C_VEL
LIN {X 0,Y 453.52,Z 327.619,A -85,B 0,C 180,E1 -8307.956,E2 -8307.956} C_VEL
LIN {X 0,Y 453.468,Z 327.627,A -85,B 0,C 180,E1 -8311.525,E2 -8311.525} C_VEL
LIN {X 0,Y 453.49,Z 327.619,A -85,B 0,C 180,E1 -8314.777,E2 -8314.777} C_VEL
LIN {X 0,Y 453.474,Z 327.62,A -85,B 0,C 180,E1 -8318.311,E2 -8318.311} C_VEL
LIN {X 0,Y 453.496,Z 327.618,A -85,B 0,C 180,E1 -8320.609,E2 -8320.609} C_VEL
LIN {X 0,Y 453.457,Z 327.627,A -85,B 0,C 180,E1 -8323.244,E2 -8323.244} C_VEL
LIN {X 0,Y 453.465,Z 327.626,A -85,B 0,C 180,E1 -8325.778,E2 -8325.778} C_VEL
LIN {X 0,Y 453.48,Z 327.62,A -85,B 0,C 180,E1 -8328.209,E2 -8328.209} C_VEL
LIN {X 0,Y 453.496,Z 327.62,A -85,B 0,C 180,E1 -8330.793,E2 -8330.793} C_VEL
LIN {X 0,Y 453.458,Z 327.628,A -85,B 0,C 180,E1 -8333.917,E2 -8333.917} C_VEL
LIN {X 0,Y 453.484,Z 327.626,A -85,B 0,C 180,E1 -8337.151,E2 -8337.151} C_VEL
LIN {X 0,Y 453.476,Z 327.623,A -85,B 0,C 180,E1 -8340.268,E2 -8340.268} C_VEL
LIN {X 0,Y 453.58,Z 327.764,A -85,B 0,C 180,E1 -8341.733,E2 -8341.733} C_VEL
LIN {X 0,Y 456.751,Z 342.672,A -85,B 0,C 180,E1 -8344.479,E2 -8344.479} C_VEL
LIN {X 0,Y 456.926,Z 346.632,A -85,B 0,C 180,E1 -8345.16,E2 -8345.16} C_VEL
LIN {X 0,Y 455.874,Z 365.54,A -85,B 0,C 180,E1 -8348.284,E2 -8348.284} C_VEL
LIN {X 0,Y 455.688,Z 368.824,A -85,B 0,C 180,E1 -8348.823,E2 -8348.823} C_VEL
LIN {X 0,Y 459.813,Z 392.537,A -85,B 0,C 180,E1 -8349.394,E2 -8349.394} C_VEL
LIN {X 0,Y 458.583,Z 506.177,A -85,B 0,C 180,E1 -8351.197,E2 -8351.197} C_VEL
LIN {X 0,Y 458.184,Z 520.392,A -85,B 0,C 180,E1 -8351.586,E2 -8351.586} C_VEL
LIN {X 0,Y 457.575,Z 534.625,A -85,B 0,C 180,E1 -8352.163,E2 -8352.163} C_VEL
LIN {X 0,Y 456.972,Z 547.369,A -85,B 0,C 180,E1 -8352.857,E2 -8352.857} C_VEL
LIN {X 0,Y 456.149,Z 560.703,A -85,B 0,C 180,E1 -8353.784,E2 -8353.784} C_VEL
LIN {X 0,Y 455.38,Z 572.324,A -85,B 0,C 180,E1 -8354.789,E2 -8354.789} C_VEL
LIN {X 0,Y 454.7,Z 582.979,A -85,B 0,C 180,E1 -8355.91,E2 -8355.91} C_VEL
LIN {X 0,Y 454.1,Z 592.915,A -85,B 0,C 180,E1 -8357.171,E2 -8357.171} C_VEL
LIN {X 0,Y 453.591,Z 602.275,A -85,B 0,C 180,E1 -8358.606,E2 -8358.606} C_VEL
LIN {X 0,Y 453.077,Z 610.63,A -85,B 0,C 180,E1 -8360.176,E2 -8360.176} C_VEL
LIN {X 0,Y 452.822,Z 616.453,A -85,B 0,C 180,E1 -8361.521,E2 -8361.521} C_VEL
LIN {X 0,Y 452.656,Z 621.241,A -85,B 0,C 180,E1 -8362.865,E2 -8362.865} C_VEL
LIN {X 0,Y 452.559,Z 626.195,A -85,B 0,C 180,E1 -8364.654,E2 -8364.654} C_VEL
LIN {X 0,Y 452.471,Z 629.641,A -85,B 0,C 180,E1 -8366.438,E2 -8366.438} C_VEL
LIN {X 0,Y 452.504,Z 630.836,A -85,B 0,C 180,E1 -8367.329,E2 -8367.329} C_VEL
LIN {X 0,Y 452.426,Z 632.201,A -85,B 0,C 180,E1 -8369.11,E2 -8369.11} C_VEL
LIN {X 0,Y 452.426,Z 632.226,A -85,B 0,C 180,E1 -8370.89,E2 -8370.89} C_VEL
LIN {X 0,Y 452.504,Z 630.911,A -85,B 0,C 180,E1 -8372.671,E2 -8372.671} C_VEL
LIN {X 0,Y 452.472,Z 628.225,A -85,B 0,C 180,E1 -8374.454,E2 -8374.454} C_VEL
LIN {X 0,Y 452.602,Z 624.104,A -85,B 0,C 180,E1 -8376.24,E2 -8376.24} C_VEL
LIN {X 0,Y 452.743,Z 618.423,A -85,B 0,C 180,E1 -8378.031,E2 -8378.031} C_VEL
LIN {X 0,Y 453.065,Z 612.03,A -85,B 0,C 180,E1 -8379.599,E2 -8379.599} C_VEL
LIN {X 0,Y 453.537,Z 604.093,A -85,B 0,C 180,E1 -8381.169,E2 -8381.169} C_VEL
LIN {X 0,Y 454.048,Z 595.006,A -85,B 0,C 180,E1 -8382.637,E2 -8382.637} C_VEL
LIN {X 0,Y 454.636,Z 585.84,A -85,B 0,C 180,E1 -8383.863,E2 -8383.863} C_VEL
LIN {X 0,Y 455.379,Z 574.774,A -85,B 0,C 180,E1 -8385.096,E2 -8385.096} C_VEL
LIN {X 0,Y 456.182,Z 563.785,A -85,B 0,C 180,E1 -8386.1,E2 -8386.1} C_VEL
LIN {X 0,Y 457.079,Z 550.63,A -85,B 0,C 180,E1 -8387.072,E2 -8387.072} C_VEL
LIN {X 0,Y 457.743,Z 537.817,A -85,B 0,C 180,E1 -8387.82,E2 -8387.82} C_VEL
LIN {X 0,Y 458.319,Z 523.861,A -85,B 0,C 180,E1 -8388.438,E2 -8388.438} C_VEL
LIN {X 0,Y 458.915,Z 509.369,A -85,B 0,C 180,E1 -8388.876,E2 -8388.876} C_VEL
LIN {X 0,Y 459.229,Z 489.159,A -85,B 0,C 180,E1 -8389.239,E2 -8389.239} C_VEL
LIN {X 0,Y 460.311,Z 392.87,A -85,B 0,C 180,E1 -8390.768,E2 -8390.768} C_VEL
LIN {X 0,Y 457.184,Z 374.924,A -85,B 0,C 180,E1 -8391.225,E2 -8391.225} C_VEL
LIN {X 0,Y 455.952,Z 368.723,A -85,B 0,C 180,E1 -8391.398,E2 -8391.398} C_VEL
LIN {X 0,Y 457.007,Z 351.466,A -85,B 0,C 180,E1 -8394.291,E2 -8394.291} C_VEL
LIN {X 0,Y 457.251,Z 344.459,A -85,B 0,C 180,E1 -8395.491,E2 -8395.491} C_VEL
LIN {X 0,Y 454.456,Z 331.638,A -85,B 0,C 180,E1 -8397.931,E2 -8397.931} C_VEL
LIN {X 0,Y 453.522,Z 327.618,A -85,B 0,C 180,E1 -8398.743,E2 -8398.743} C_VEL
LIN {X 0,Y 453.466,Z 327.622,A -85,B 0,C 180,E1 -8401.8,E2 -8401.8} C_VEL
LIN {X 0,Y 453.482,Z 327.624,A -85,B 0,C 180,E1 -8404.989,E2 -8404.989} C_VEL
LIN {X 0,Y 453.465,Z 327.621,A -85,B 0,C 180,E1 -8408.312,E2 -8408.312} C_VEL
LIN {X 0,Y 453.495,Z 327.623,A -85,B 0,C 180,E1 -8410.609,E2 -8410.609} C_VEL
LIN {X 0,Y 453.454,Z 327.621,A -85,B 0,C 180,E1 -8413.244,E2 -8413.244} C_VEL
LIN {X 0,Y 453.465,Z 327.621,A -85,B 0,C 180,E1 -8415.779,E2 -8415.779} C_VEL
LIN {X 0,Y 453.481,Z 327.622,A -85,B 0,C 180,E1 -8418.21,E2 -8418.21} C_VEL
LIN {X 0,Y 453.517,Z 327.616,A -85,B 0,C 180,E1 -8420.79,E2 -8420.79} C_VEL
LIN {X 0,Y 453.454,Z 327.623,A -85,B 0,C 180,E1 -8423.917,E2 -8423.917} C_VEL
LIN {X 0,Y 453.486,Z 327.617,A -85,B 0,C 180,E1 -8427.152,E2 -8427.152} C_VEL
LIN {X 0,Y 453.47,Z 327.623,A -85,B 0,C 180,E1 -8430.268,E2 -8430.268} C_VEL
LIN {X 0,Y 453.474,Z 327.618,A -85,B 0,C 180,E1 -8433.292,E2 -8433.292} C_VEL
LIN {X 0,Y 453.5,Z 327.622,A -85,B 0,C 180,E1 -8436.239,E2 -8436.239} C_VEL
LIN {X 0,Y 453.486,Z 327.617,A -85,B 0,C 180,E1 -8439.118,E2 -8439.118} C_VEL
LIN {X 0,Y 453.506,Z 327.618,A -85,B 0,C 180,E1 -8441.945,E2 -8441.945} C_VEL
LIN {X 0,Y 453.543,Z 327.612,A -85,B 0,C 180,E1 -8444.727,E2 -8444.727} C_VEL
LIN {X 0,Y 453.562,Z 327.612,A -85,B 0,C 180,E1 -8448.379,E2 -8448.379} C_VEL
LIN {X 0,Y 453.586,Z 327.603,A -85,B 0,C 180,E1 -8451.087,E2 -8451.087} C_VEL
LIN {X 0,Y 453.646,Z 327.602,A -85,B 0,C 180,E1 -8453.775,E2 -8453.775} C_VEL
LIN {X 0,Y 453.709,Z 327.586,A -85,B 0,C 180,E1 -8457.337,E2 -8457.337} C_VEL
LIN {X 0,Y 453.793,Z 327.584,A -85,B 0,C 180,E1 -8460,E2 -8460} C_VEL
LIN {X 0,Y 453.736,Z 327.585,A -85,B 0,C 180,E1 -8462.664,E2 -8462.664} C_VEL
LIN {X 0,Y 453.639,Z 327.595,A -85,B 0,C 180,E1 -8466.226,E2 -8466.226} C_VEL
LIN {X 0,Y 453.582,Z 327.606,A -85,B 0,C 180,E1 -8468.914,E2 -8468.914} C_VEL
LIN {X 0,Y 453.568,Z 327.606,A -85,B 0,C 180,E1 -8472.529,E2 -8472.529} C_VEL
LIN {X 0,Y 453.502,Z 327.614,A -85,B 0,C 180,E1 -8476.089,E2 -8476.089} C_VEL
LIN {X 0,Y 453.489,Z 327.619,A -85,B 0,C 180,E1 -8479.028,E2 -8479.028} C_VEL
LIN {X 0,Y 453.475,Z 327.625,A -85,B 0,C 180,E1 -8481.837,E2 -8481.837} C_VEL
LIN {X 0,Y 453.473,Z 327.617,A -85,B 0,C 180,E1 -8484.737,E2 -8484.737} C_VEL
LIN {X 0,Y 453.461,Z 327.62,A -85,B 0,C 180,E1 -8487.942,E2 -8487.942} C_VEL
LIN {X 0,Y 453.45,Z 327.608,A -85,B 0,C 180,E1 -8490.762,E2 -8490.762} C_VEL
LIN {X 0,Y 453.468,Z 327.622,A -85,B 0,C 180,E1 -8493.914,E2 -8493.914} C_VEL
LIN {X 0,Y 453.436,Z 327.617,A -85,B 0,C 180,E1 -8497.192,E2 -8497.192} C_VEL
LIN {X 0,Y 453.467,Z 327.619,A -85,B 0,C 180,E1 -8500.612,E2 -8500.612} C_VEL
LIN {X 0,Y 453.479,Z 327.621,A -85,B 0,C 180,E1 -8504.528,E2 -8504.528} C_VEL
LIN {X 0,Y 453.433,Z 327.628,A -85,B 0,C 180,E1 -8508.072,E2 -8508.072} C_VEL
LIN {X 0,Y 453.425,Z 327.631,A -85,B 0,C 180,E1 -8510.805,E2 -8510.805} C_VEL
LIN {X 0,Y 453.44,Z 327.627,A -85,B 0,C 180,E1 -8513.916,E2 -8513.916} C_VEL
LIN {X 0,Y 453.468,Z 327.623,A -85,B 0,C 180,E1 -8516.816,E2 -8516.816} C_VEL
LIN {X 0,Y 453.46,Z 327.703,A -85,B 0,C 180,E1 -8519.896,E2 -8519.896} C_VEL
LIN {X 0,Y 455.967,Z 339.535,A -85,B 0,C 180,E1 -8522.458,E2 -8522.458} C_VEL
LIN {X 0,Y 456.31,Z 343.642,A -85,B 0,C 180,E1 -8523.293,E2 -8523.293} C_VEL
LIN {X 0,Y 456.196,Z 345.689,A -85,B 0,C 180,E1 -8523.674,E2 -8523.674} C_VEL
LIN {X 0,Y 460.492,Z 364.881,A -85,B 0,C 180,E1 -8524.219,E2 -8524.219} C_VEL
LIN {X 0,Y 459.468,Z 467.007,A -85,B 0,C 180,E1 -8525.849,E2 -8525.849} C_VEL
LIN {X 0,Y 458.677,Z 472.87,A -85,B 0,C 180,E1 -8525.907,E2 -8525.907} C_VEL
LIN {X 0,Y 455.689,Z 482.376,A -85,B 0,C 180,E1 -8525.947,E2 -8525.947} C_VEL
LIN {X 0,Y 452.811,Z 491.779,A -85,B 0,C 180,E1 -8526.069,E2 -8526.069} C_VEL
LIN {X 0,Y 452.13,Z 497.46,A -85,B 0,C 180,E1 -8526.24,E2 -8526.24} C_VEL
LIN {X 0,Y 451.527,Z 509.78,A -85,B 0,C 180,E1 -8526.755,E2 -8526.755} C_VEL
LIN {X 0,Y 450.941,Z 522.003,A -85,B 0,C 180,E1 -8527.431,E2 -8527.431} C_VEL
LIN {X 0,Y 450.073,Z 535.087,A -85,B 0,C 180,E1 -8528.351,E2 -8528.351} C_VEL
LIN {X 0,Y 449.28,Z 546.913,A -85,B 0,C 180,E1 -8529.392,E2 -8529.392} C_VEL
LIN {X 0,Y 448.46,Z 558.04,A -85,B 0,C 180,E1 -8530.589,E2 -8530.589} C_VEL
LIN {X 0,Y 447.669,Z 568.352,A -85,B 0,C 180,E1 -8531.937,E2 -8531.937} C_VEL
LIN {X 0,Y 447.044,Z 577.105,A -85,B 0,C 180,E1 -8533.327,E2 -8533.327} C_VEL
LIN {X 0,Y 446.448,Z 585.463,A -85,B 0,C 180,E1 -8534.945,E2 -8534.945} C_VEL
LIN {X 0,Y 446.065,Z 591.26,A -85,B 0,C 180,E1 -8536.33,E2 -8536.33} C_VEL
LIN {X 0,Y 445.713,Z 596.462,A -85,B 0,C 180,E1 -8537.857,E2 -8537.857} C_VEL
LIN {X 0,Y 445.563,Z 600.904,A -85,B 0,C 180,E1 -8539.549,E2 -8539.549} C_VEL
LIN {X 0,Y 445.416,Z 603.565,A -85,B 0,C 180,E1 -8540.922,E2 -8540.922} C_VEL
LIN {X 0,Y 445.387,Z 605.872,A -85,B 0,C 180,E1 -8542.748,E2 -8542.748} C_VEL
LIN {X 0,Y 445.396,Z 606.833,A -85,B 0,C 180,E1 -8544.567,E2 -8544.567} C_VEL
LIN {X 0,Y 445.359,Z 606.476,A -85,B 0,C 180,E1 -8546.381,E2 -8546.381} C_VEL
LIN {X 0,Y 445.4,Z 604.8,A -85,B 0,C 180,E1 -8548.192,E2 -8548.192} C_VEL
LIN {X 0,Y 445.436,Z 601.779,A -85,B 0,C 180,E1 -8550,E2 -8550} C_VEL
LIN {X 0,Y 445.588,Z 597.328,A -85,B 0,C 180,E1 -8551.808,E2 -8551.808} C_VEL
LIN {X 0,Y 445.919,Z 592.906,A -85,B 0,C 180,E1 -8553.162,E2 -8553.162} C_VEL
LIN {X 0,Y 446.242,Z 587.542,A -85,B 0,C 180,E1 -8554.517,E2 -8554.517} C_VEL
LIN {X 0,Y 446.784,Z 579.874,A -85,B 0,C 180,E1 -8556.095,E2 -8556.095} C_VEL
LIN {X 0,Y 447.301,Z 572.081,A -85,B 0,C 180,E1 -8557.418,E2 -8557.418} C_VEL
LIN {X 0,Y 447.773,Z 564.037,A -85,B 0,C 180,E1 -8558.575,E2 -8558.575} C_VEL
LIN {X 0,Y 448.634,Z 552.658,A -85,B 0,C 180,E1 -8559.923,E2 -8559.923} C_VEL
LIN {X 0,Y 449.328,Z 541.08,A -85,B 0,C 180,E1 -8561.046,E2 -8561.046} C_VEL
LIN {X 0,Y 450.134,Z 528.202,A -85,B 0,C 180,E1 -8562.054,E2 -8562.054} C_VEL
LIN {X 0,Y 450.904,Z 514.558,A -85,B 0,C 180,E1 -8562.89,E2 -8562.89} C_VEL
LIN {X 0,Y 451.47,Z 500.58,A -85,B 0,C 180,E1 -8563.532,E2 -8563.532} C_VEL
LIN {X 0,Y 451.83,Z 486.832,A -85,B 0,C 180,E1 -8563.98,E2 -8563.98} C_VEL
LIN {X 0,Y 452.129,Z 469.619,A -85,B 0,C 180,E1 -8564.315,E2 -8564.315} C_VEL
LIN {X 0,Y 453.252,Z 365.466,A -85,B 0,C 180,E1 -8565.979,E2 -8565.979} C_VEL
LIN {X 0,Y 449.025,Z 345.697,A -85,B 0,C 180,E1 -8566.503,E2 -8566.503} C_VEL
LIN {X 0,Y 449.074,Z 341.524,A -85,B 0,C 180,E1 -8567.32,E2 -8567.32} C_VEL
LIN {X 0,Y 446.44,Z 328.503,A -85,B 0,C 180,E1 -8570.083,E2 -8570.083} C_VEL
LIN {X 0,Y 446.413,Z 328.506,A -85,B 0,C 180,E1 -8573.178,E2 -8573.178} C_VEL
LIN {X 0,Y 446.419,Z 328.503,A -85,B 0,C 180,E1 -8576.187,E2 -8576.187} C_VEL
LIN {X 0,Y 446.411,Z 328.502,A -85,B 0,C 180,E1 -8579.212,E2 -8579.212} C_VEL
LIN {X 0,Y 446.399,Z 328.505,A -85,B 0,C 180,E1 -8582.364,E2 -8582.364} C_VEL
LIN {X 0,Y 446.408,Z 328.501,A -85,B 0,C 180,E1 -8585.627,E2 -8585.627} C_VEL
LIN {X 0,Y 446.388,Z 328.506,A -85,B 0,C 180,E1 -8589.033,E2 -8589.033} C_VEL
LIN {X 0,Y 446.379,Z 328.505,A -85,B 0,C 180,E1 -8592.269,E2 -8592.269} C_VEL
LIN {X 0,Y 446.424,Z 328.499,A -85,B 0,C 180,E1 -8595.108,E2 -8595.108} C_VEL
LIN {X 0,Y 446.398,Z 328.504,A -85,B 0,C 180,E1 -8598.605,E2 -8598.605} C_VEL
LIN {X 0,Y 446.39,Z 328.504,A -85,B 0,C 180,E1 -8602.119,E2 -8602.119} C_VEL
LIN {X 0,Y 446.423,Z 328.498,A -85,B 0,C 180,E1 -8605.476,E2 -8605.476} C_VEL
LIN {X 0,Y 446.394,Z 328.507,A -85,B 0,C 180,E1 -8608.697,E2 -8608.697} C_VEL
LIN {X 0,Y 446.405,Z 328.499,A -85,B 0,C 180,E1 -8611.841,E2 -8611.841} C_VEL
LIN {X 0,Y 446.424,Z 328.5,A -85,B 0,C 180,E1 -8614.845,E2 -8614.845} C_VEL
LIN {X 0,Y 446.45,Z 328.491,A -85,B 0,C 180,E1 -8618.246,E2 -8618.246} C_VEL
LIN {X 0,Y 446.442,Z 328.489,A -85,B 0,C 180,E1 -8621.648,E2 -8621.648} C_VEL
LIN {X 0,Y 446.461,Z 328.498,A -85,B 0,C 180,E1 -8624.478,E2 -8624.478} C_VEL
LIN {X 0,Y 446.52,Z 328.478,A -85,B 0,C 180,E1 -8627.384,E2 -8627.384} C_VEL
LIN {X 0,Y 446.534,Z 328.479,A -85,B 0,C 180,E1 -8630.944,E2 -8630.944} C_VEL
LIN {X 0,Y 446.612,Z 328.476,A -85,B 0,C 180,E1 -8633.676,E2 -8633.676} C_VEL
LIN {X 0,Y 446.683,Z 328.464,A -85,B 0,C 180,E1 -8637.294,E2 -8637.294} C_VEL
LIN {X 0,Y 446.741,Z 328.463,A -85,B 0,C 180,E1 -8640,E2 -8640} C_VEL
LIN {X 0,Y 446.658,Z 328.47,A -85,B 0,C 180,E1 -8642.705,E2 -8642.705} C_VEL
LIN {X 0,Y 446.614,Z 328.477,A -85,B 0,C 180,E1 -8646.324,E2 -8646.324} C_VEL
LIN {X 0,Y 446.533,Z 328.483,A -85,B 0,C 180,E1 -8649.055,E2 -8649.055} C_VEL
LIN {X 0,Y 446.525,Z 328.485,A -85,B 0,C 180,E1 -8652.729,E2 -8652.729} C_VEL
LIN {X 0,Y 446.499,Z 328.492,A -85,B 0,C 180,E1 -8656.227,E2 -8656.227} C_VEL
LIN {X 0,Y 446.471,Z 328.492,A -85,B 0,C 180,E1 -8659.303,E2 -8659.303} C_VEL
LIN {X 0,Y 446.421,Z 328.5,A -85,B 0,C 180,E1 -8662.199,E2 -8662.199} C_VEL
LIN {X 0,Y 446.443,Z 328.497,A -85,B 0,C 180,E1 -8665.153,E2 -8665.153} C_VEL
LIN {X 0,Y 446.487,Z 328.492,A -85,B 0,C 180,E1 -8668.178,E2 -8668.178} C_VEL
LIN {X 0,Y 446.422,Z 328.504,A -85,B 0,C 180,E1 -8671.775,E2 -8671.775} C_VEL
LIN {X 0,Y 446.431,Z 328.499,A -85,B 0,C 180,E1 -8674.523,E2 -8674.523} C_VEL
LIN {X 0,Y 446.432,Z 328.499,A -85,B 0,C 180,E1 -8678.081,E2 -8678.081} C_VEL
LIN {X 0,Y 446.429,Z 328.5,A -85,B 0,C 180,E1 -8680.917,E2 -8680.917} C_VEL
LIN {X 0,Y 446.402,Z 328.506,A -85,B 0,C 180,E1 -8683.846,E2 -8683.846} C_VEL
LIN {X 0,Y 446.399,Z 328.501,A -85,B 0,C 180,E1 -8686.403,E2 -8686.403} C_VEL
LIN {X 0,Y 446.428,Z 328.501,A -85,B 0,C 180,E1 -8689.082,E2 -8689.082} C_VEL
LIN {X 0,Y 446.429,Z 328.502,A -85,B 0,C 180,E1 -8692.123,E2 -8692.123} C_VEL
LIN {X 0,Y 446.432,Z 328.506,A -85,B 0,C 180,E1 -8695.477,E2 -8695.477} C_VEL
LIN {X 0,Y 446.417,Z 328.503,A -85,B 0,C 180,E1 -8698.7,E2 -8698.7} C_VEL
LIN {X 0,Y 446.507,Z 328.564,A -85,B 0,C 180,E1 -8701.452,E2 -8701.452} C_VEL
LIN {X 0,Y 449.769,Z 343.754,A -85,B 0,C 180,E1 -8704.303,E2 -8704.303} C_VEL
LIN {X 0,Y 450.073,Z 347.217,A -85,B 0,C 180,E1 -8704.916,E2 -8704.916} C_VEL
LIN {X 0,Y 448.936,Z 366.614,A -85,B 0,C 180,E1 -8708.173,E2 -8708.173} C_VEL
LIN {X 0,Y 448.796,Z 368.605,A -85,B 0,C 180,E1 -8708.504,E2 -8708.504} C_VEL
LIN {X 0,Y 453.103,Z 393.206,A -85,B 0,C 180,E1 -8709.113,E2 -8709.113} C_VEL
LIN {X 0,Y 451.804,Z 506.313,A -85,B 0,C 180,E1 -8710.934,E2 -8710.934} C_VEL
LIN {X 0,Y 451.359,Z 521.152,A -85,B 0,C 180,E1 -8711.356,E2 -8711.356} C_VEL
LIN {X 0,Y 450.784,Z 534.221,A -85,B 0,C 180,E1 -8711.897,E2 -8711.897} C_VEL
LIN {X 0,Y 450.11,Z 547.123,A -85,B 0,C 180,E1 -8712.606,E2 -8712.606} C_VEL
LIN {X 0,Y 449.254,Z 560.239,A -85,B 0,C 180,E1 -8713.528,E2 -8713.528} C_VEL
LIN {X 0,Y 448.487,Z 571.912,A -85,B 0,C 180,E1 -8714.55,E2 -8714.55} C_VEL
LIN {X 0,Y 447.763,Z 582.606,A -85,B 0,C 180,E1 -8715.688,E2 -8715.688} C_VEL
LIN {X 0,Y 447.063,Z 593.35,A -85,B 0,C 180,E1 -8717.075,E2 -8717.075} C_VEL
LIN {X 0,Y 446.483,Z 603.273,A -85,B 0,C 180,E1 -8718.652,E2 -8718.652} C_VEL
LIN {X 0,Y 445.978,Z 611.367,A -85,B 0,C 180,E1 -8720.247,E2 -8720.247} C_VEL
LIN {X 0,Y 445.663,Z 617.886,A -85,B 0,C 180,E1 -8721.841,E2 -8721.841} C_VEL
LIN {X 0,Y 445.528,Z 623.666,A -85,B 0,C 180,E1 -8723.66,E2 -8723.66} C_VEL
LIN {X 0,Y 445.394,Z 627.862,A -85,B 0,C 180,E1 -8725.475,E2 -8725.475} C_VEL
LIN {X 0,Y 445.428,Z 630.614,A -85,B 0,C 180,E1 -8727.287,E2 -8727.287} C_VEL
LIN {X 0,Y 445.336,Z 631.991,A -85,B 0,C 180,E1 -8729.096,E2 -8729.096} C_VEL
LIN {X 0,Y 445.336,Z 632.03,A -85,B 0,C 180,E1 -8730.904,E2 -8730.904} C_VEL
LIN {X 0,Y 445.428,Z 630.73,A -85,B 0,C 180,E1 -8732.713,E2 -8732.713} C_VEL
LIN {X 0,Y 445.395,Z 628.057,A -85,B 0,C 180,E1 -8734.525,E2 -8734.525} C_VEL
LIN {X 0,Y 445.528,Z 623.949,A -85,B 0,C 180,E1 -8736.34,E2 -8736.34} C_VEL
LIN {X 0,Y 445.688,Z 618.285,A -85,B 0,C 180,E1 -8738.159,E2 -8738.159} C_VEL
LIN {X 0,Y 446.022,Z 611.91,A -85,B 0,C 180,E1 -8739.752,E2 -8739.752} C_VEL
LIN {X 0,Y 446.512,Z 603.994,A -85,B 0,C 180,E1 -8741.347,E2 -8741.347} C_VEL
LIN {X 0,Y 447.02,Z 595.73,A -85,B 0,C 180,E1 -8742.715,E2 -8742.715} C_VEL
LIN {X 0,Y 447.701,Z 585.795,A -85,B 0,C 180,E1 -8744.083,E2 -8744.083} C_VEL
LIN {X 0,Y 448.506,Z 574.765,A -85,B 0,C 180,E1 -8745.333,E2 -8745.333} C_VEL
LIN {X 0,Y 449.514,Z 562.473,A -85,B 0,C 180,E1 -8746.462,E2 -8746.462} C_VEL
LIN {X 0,Y 450.294,Z 550.839,A -85,B 0,C 180,E1 -8747.332,E2 -8747.332} C_VEL
LIN {X 0,Y 450.991,Z 538.235,A -85,B 0,C 180,E1 -8748.086,E2 -8748.086} C_VEL
LIN {X 0,Y 451.624,Z 524.238,A -85,B 0,C 180,E1 -8748.721,E2 -8748.721} C_VEL
LIN {X 0,Y 452.241,Z 510.037,A -85,B 0,C 180,E1 -8749.165,E2 -8749.165} C_VEL
LIN {X 0,Y 452.58,Z 490.329,A -85,B 0,C 180,E1 -8749.533,E2 -8749.533} C_VEL
LIN {X 0,Y 453.639,Z 392.73,A -85,B 0,C 180,E1 -8751.111,E2 -8751.111} C_VEL
LIN {X 0,Y 449.932,Z 372.552,A -85,B 0,C 180,E1 -8751.648,E2 -8751.648} C_VEL
LIN {X 0,Y 449.154,Z 368.354,A -85,B 0,C 180,E1 -8751.792,E2 -8751.792} C_VEL
LIN {X 0,Y 450.244,Z 351.43,A -85,B 0,C 180,E1 -8754.68,E2 -8754.68} C_VEL
LIN {X 0,Y 450.499,Z 346.898,A -85,B 0,C 180,E1 -8755.464,E2 -8755.464} C_VEL
LIN {X 0,Y 448.286,Z 336.038,A -85,B 0,C 180,E1 -8757.548,E2 -8757.548} C_VEL
LIN {X 0,Y 446.488,Z 328.493,A -85,B 0,C 180,E1 -8759.085,E2 -8759.085} C_VEL
LIN {X 0,Y 446.424,Z 328.501,A -85,B 0,C 180,E1 -8762.362,E2 -8762.362} C_VEL
LIN {X 0,Y 446.421,Z 328.501,A -85,B 0,C 180,E1 -8765.626,E2 -8765.626} C_VEL
LIN {X 0,Y 446.443,Z 328.496,A -85,B 0,C 180,E1 -8769.028,E2 -8769.028} C_VEL
LIN {X 0,Y 446.436,Z 328.501,A -85,B 0,C 180,E1 -8772.278,E2 -8772.278} C_VEL
LIN {X 0,Y 446.453,Z 328.494,A -85,B 0,C 180,E1 -8775.104,E2 -8775.104} C_VEL
LIN {X 0,Y 446.43,Z 328.502,A -85,B 0,C 180,E1 -8778.609,E2 -8778.609} C_VEL
LIN {X 0,Y 446.461,Z 328.493,A -85,B 0,C 180,E1 -8780.975,E2 -8780.975} C_VEL
LIN {X 0,Y 446.42,Z 328.503,A -85,B 0,C 180,E1 -8784.374,E2 -8784.374} C_VEL
LIN {X 0,Y 446.425,Z 328.497,A -85,B 0,C 180,E1 -8787.639,E2 -8787.639} C_VEL
LIN {X 0,Y 446.44,Z 328.497,A -85,B 0,C 180,E1 -8790.79,E2 -8790.79} C_VEL
LIN {X 0,Y 446.442,Z 328.497,A -85,B 0,C 180,E1 -8793.846,E2 -8793.846} C_VEL
LIN {X 0,Y 446.429,Z 328.496,A -85,B 0,C 180,E1 -8796.824,E2 -8796.824} C_VEL
LIN {X 0,Y 446.447,Z 328.497,A -85,B 0,C 180,E1 -8799.737,E2 -8799.737} C_VEL
LIN {X 0,Y 446.459,Z 328.493,A -85,B 0,C 180,E1 -8802.597,E2 -8802.597} C_VEL
LIN {X 0,Y 446.473,Z 328.493,A -85,B 0,C 180,E1 -8805.413,E2 -8805.413} C_VEL
LIN {X 0,Y 446.521,Z 328.491,A -85,B 0,C 180,E1 -8808.193,E2 -8808.193} C_VEL
LIN {X 0,Y 446.534,Z 328.481,A -85,B 0,C 180,E1 -8810.945,E2 -8810.945} C_VEL
LIN {X 0,Y 446.615,Z 328.477,A -85,B 0,C 180,E1 -8813.676,E2 -8813.676} C_VEL
LIN {X 0,Y 446.658,Z 328.464,A -85,B 0,C 180,E1 -8817.295,E2 -8817.295} C_VEL
LIN {X 0,Y 446.741,Z 328.462,A -85,B 0,C 180,E1 -8820,E2 -8820} C_VEL
LIN {X 0,Y 446.683,Z 328.463,A -85,B 0,C 180,E1 -8822.706,E2 -8822.706} C_VEL
LIN {X 0,Y 446.609,Z 328.47,A -85,B 0,C 180,E1 -8826.325,E2 -8826.325} C_VEL
LIN {X 0,Y 446.53,Z 328.485,A -85,B 0,C 180,E1 -8829.056,E2 -8829.056} C_VEL
LIN {X 0,Y 446.526,Z 328.483,A -85,B 0,C 180,E1 -8832.73,E2 -8832.73} C_VEL
LIN {X 0,Y 446.454,Z 328.491,A -85,B 0,C 180,E1 -8836.207,E2 -8836.207} C_VEL
LIN {X 0,Y 446.435,Z 328.5,A -85,B 0,C 180,E1 -8839.305,E2 -8839.305} C_VEL
LIN {X 0,Y 446.415,Z 328.501,A -85,B 0,C 180,E1 -8842.2,E2 -8842.2} C_VEL
LIN {X 0,Y 446.425,Z 328.497,A -85,B 0,C 180,E1 -8845.155,E2 -8845.155} C_VEL
LIN {X 0,Y 446.419,Z 328.496,A -85,B 0,C 180,E1 -8848.184,E2 -8848.184} C_VEL
LIN {X 0,Y 446.394,Z 328.492,A -85,B 0,C 180,E1 -8851.303,E2 -8851.303} C_VEL
LIN {X 0,Y 446.423,Z 328.498,A -85,B 0,C 180,E1 -8854.524,E2 -8854.524} C_VEL
LIN {X 0,Y 446.396,Z 328.502,A -85,B 0,C 180,E1 -8858.075,E2 -8858.075} C_VEL
LIN {X 0,Y 446.398,Z 328.508,A -85,B 0,C 180,E1 -8861.395,E2 -8861.395} C_VEL
LIN {X 0,Y 446.423,Z 328.5,A -85,B 0,C 180,E1 -8865.108,E2 -8865.108} C_VEL
LIN {X 0,Y 446.398,Z 328.505,A -85,B 0,C 180,E1 -8868.605,E2 -8868.605} C_VEL
LIN {X 0,Y 446.388,Z 328.506,A -85,B 0,C 180,E1 -8872.119,E2 -8872.119} C_VEL
LIN {X 0,Y 446.415,Z 328.505,A -85,B 0,C 180,E1 -8875.475,E2 -8875.475} C_VEL
LIN {X 0,Y 446.392,Z 328.506,A -85,B 0,C 180,E1 -8878.697,E2 -8878.697} C_VEL
LIN {X 0,Y 446.427,Z 328.592,A -85,B 0,C 180,E1 -8879.587,E2 -8879.587} C_VEL
LIN {X 0,Y 448.991,Z 340.66,A -85,B 0,C 180,E1 -8882.246,E2 -8882.246} C_VEL
LIN {X 0,Y 449.439,Z 344.47,A -85,B 0,C 180,E1 -8883.041,E2 -8883.041} C_VEL
LIN {X 0,Y 449.365,Z 345.805,A -85,B 0,C 180,E1 -8883.305,E2 -8883.305} C_VEL
LIN {X 0,Y 453.939,Z 365.884,A -85,B 0,C 180,E1 -8883.894,E2 -8883.894} C_VEL
LIN {X 0,Y 452.642,Z 482.132,A -85,B 0,C 180,E1 -8885.795,E2 -8885.795} C_VEL
LIN {X 0,Y 452.169,Z 496.623,A -85,B 0,C 180,E1 -8886.209,E2 -8886.209} C_VEL
LIN {X 0,Y 452.13,Z 497.46,A -85,B 0,C 180,E1 -8886.24,E2 -8886.24} C_VEL
LIN {X 0,Y 451.365,Z 503.24,A -85,B 0,C 180,E1 -8886.438,E2 -8886.438} C_VEL
LIN {X 0,Y 448.19,Z 512.424,A -85,B 0,C 180,E1 -8886.737,E2 -8886.737} C_VEL
LIN {X 0,Y 444.906,Z 521.265,A -85,B 0,C 180,E1 -8887.101,E2 -8887.101} C_VEL
LIN {X 0,Y 443.972,Z 526.434,A -85,B 0,C 180,E1 -8887.409,E2 -8887.409} C_VEL
LIN {X 0,Y 443.105,Z 538.885,A -85,B 0,C 180,E1 -8888.36,E2 -8888.36} C_VEL
LIN {X 0,Y 442.291,Z 550.062,A -85,B 0,C 180,E1 -8889.417,E2 -8889.417} C_VEL
LIN {X 0,Y 441.358,Z 561.246,A -85,B 0,C 180,E1 -8890.706,E2 -8890.706} C_VEL
LIN {X 0,Y 440.533,Z 571.262,A -85,B 0,C 180,E1 -8892.115,E2 -8892.115} C_VEL
LIN {X 0,Y 439.905,Z 579.836,A -85,B 0,C 180,E1 -8893.582,E2 -8893.582} C_VEL
LIN {X 0,Y 439.298,Z 587.436,A -85,B 0,C 180,E1 -8895.169,E2 -8895.169} C_VEL
LIN {X 0,Y 438.959,Z 592.94,A -85,B 0,C 180,E1 -8896.576,E2 -8896.576} C_VEL
LIN {X 0,Y 438.575,Z 598.695,A -85,B 0,C 180,E1 -8898.445,E2 -8898.445} C_VEL
LIN {X 0,Y 438.413,Z 601.972,A -85,B 0,C 180,E1 -8899.843,E2 -8899.843} C_VEL
LIN {X 0,Y 438.299,Z 605.019,A -85,B 0,C 180,E1 -8901.702,E2 -8901.702} C_VEL
LIN {X 0,Y 438.319,Z 606.688,A -85,B 0,C 180,E1 -8903.556,E2 -8903.556} C_VEL
LIN {X 0,Y 438.279,Z 607.031,A -85,B 0,C 180,E1 -8905.401,E2 -8905.401} C_VEL
LIN {X 0,Y 438.363,Z 606.054,A -85,B 0,C 180,E1 -8907.243,E2 -8907.243} C_VEL
LIN {X 0,Y 438.287,Z 603.758,A -85,B 0,C 180,E1 -8909.081,E2 -8909.081} C_VEL
LIN {X 0,Y 438.422,Z 600.077,A -85,B 0,C 180,E1 -8910.918,E2 -8910.918} C_VEL
LIN {X 0,Y 438.674,Z 594.905,A -85,B 0,C 180,E1 -8912.755,E2 -8912.755} C_VEL
LIN {X 0,Y 439.137,Z 589.883,A -85,B 0,C 180,E1 -8914.13,E2 -8914.13} C_VEL
LIN {X 0,Y 439.592,Z 582.739,A -85,B 0,C 180,E1 -8915.735,E2 -8915.735} C_VEL
LIN {X 0,Y 440.17,Z 573.924,A -85,B 0,C 180,E1 -8917.339,E2 -8917.339} C_VEL
LIN {X 0,Y 440.786,Z 564.686,A -85,B 0,C 180,E1 -8918.712,E2 -8918.712} C_VEL
LIN {X 0,Y 441.689,Z 553.394,A -85,B 0,C 180,E1 -8920.08,E2 -8920.08} C_VEL
LIN {X 0,Y 442.416,Z 541.923,A -85,B 0,C 180,E1 -8921.221,E2 -8921.221} C_VEL
LIN {X 0,Y 443.264,Z 529.184,A -85,B 0,C 180,E1 -8922.243,E2 -8922.243} C_VEL
LIN {X 0,Y 444.007,Z 516.735,A -85,B 0,C 180,E1 -8923.036,E2 -8923.036} C_VEL
LIN {X 0,Y 444.648,Z 502.872,A -85,B 0,C 180,E1 -8923.715,E2 -8923.715} C_VEL
LIN {X 0,Y 445.096,Z 489.16,A -85,B 0,C 180,E1 -8924.196,E2 -8924.196} C_VEL
LIN {X 0,Y 445.36,Z 475.067,A -85,B 0,C 180,E1 -8924.508,E2 -8924.508} C_VEL
LIN {X 0,Y 446.594,Z 366.411,A -85,B 0,C 180,E1 -8926.268,E2 -8926.268} C_VEL
LIN {X 0,Y 442.169,Z 345.816,A -85,B 0,C 180,E1 -8926.841,E2 -8926.841} C_VEL
LIN {X 0,Y 442.006,Z 342.138,A -85,B 0,C 180,E1 -8927.584,E2 -8927.584} C_VEL
LIN {X 0,Y 439.415,Z 329.379,A -85,B 0,C 180,E1 -8930.357,E2 -8930.357} C_VEL
LIN {X 0,Y 439.359,Z 329.383,A -85,B 0,C 180,E1 -8933.572,E2 -8933.572} C_VEL
LIN {X 0,Y 439.358,Z 329.386,A -85,B 0,C 180,E1 -8936.609,E2 -8936.609} C_VEL
LIN {X 0,Y 439.36,Z 329.377,A -85,B 0,C 180,E1 -8939.728,E2 -8939.728} C_VEL
LIN {X 0,Y 439.344,Z 329.385,A -85,B 0,C 180,E1 -8942.949,E2 -8942.949} C_VEL
LIN {X 0,Y 439.365,Z 329.38,A -85,B 0,C 180,E1 -8946.288,E2 -8946.288} C_VEL
LIN {X 0,Y 439.35,Z 329.386,A -85,B 0,C 180,E1 -8948.599,E2 -8948.599} C_VEL
LIN {X 0,Y 439.347,Z 329.38,A -85,B 0,C 180,E1 -8952.21,E2 -8952.21} C_VEL
LIN {X 0,Y 439.378,Z 329.375,A -85,B 0,C 180,E1 -8955.267,E2 -8955.267} C_VEL
LIN {X 0,Y 439.35,Z 329.381,A -85,B 0,C 180,E1 -8959.015,E2 -8959.015} C_VEL
LIN {X 0,Y 439.335,Z 329.383,A -85,B 0,C 180,E1 -8962.563,E2 -8962.563} C_VEL
LIN {X 0,Y 439.394,Z 329.377,A -85,B 0,C 180,E1 -8964.843,E2 -8964.843} C_VEL
LIN {X 0,Y 439.356,Z 329.376,A -85,B 0,C 180,E1 -8968.138,E2 -8968.138} C_VEL
LIN {X 0,Y 439.388,Z 329.372,A -85,B 0,C 180,E1 -8971.61,E2 -8971.61} C_VEL
LIN {X 0,Y 439.37,Z 329.381,A -85,B 0,C 180,E1 -8974.413,E2 -8974.413} C_VEL
LIN {X 0,Y 439.363,Z 329.374,A -85,B 0,C 180,E1 -8977.424,E2 -8977.424} C_VEL
LIN {X 0,Y 439.444,Z 329.361,A -85,B 0,C 180,E1 -8980.663,E2 -8980.663} C_VEL
LIN {X 0,Y 439.42,Z 329.376,A -85,B 0,C 180,E1 -8984.223,E2 -8984.223} C_VEL
LIN {X 0,Y 439.488,Z 329.354,A -85,B 0,C 180,E1 -8987.285,E2 -8987.285} C_VEL
LIN {X 0,Y 439.498,Z 329.356,A -85,B 0,C 180,E1 -8990.798,E2 -8990.798} C_VEL
LIN {X 0,Y 439.564,Z 329.353,A -85,B 0,C 180,E1 -8993.574,E2 -8993.574} C_VEL
LIN {X 0,Y 439.419,Z 329.37,A -85,B 0,C 180,E1 -8995.413,E2 -8995.413} C_VEL
LIN {X 0,Y 439.636,Z 329.35,A -85,B 0,C 180,E1 -8998.168,E2 -8998.168} C_VEL
LIN {X 0,Y 439.589,Z 329.345,A -85,B 0,C 180,E1 -9000.916,E2 -9000.916} C_VEL
LIN {X 0,Y 439.61,Z 329.347,A -85,B 0,C 180,E1 -9002.749,E2 -9002.749} C_VEL
LIN {X 0,Y 439.607,Z 329.346,A -85,B 0,C 180,E1 -9005.504,E2 -9005.504} C_VEL
LIN {X 0,Y 439.506,Z 329.363,A -85,B 0,C 180,E1 -9008.274,E2 -9008.274} C_VEL
LIN {X 0,Y 439.486,Z 329.369,A -85,B 0,C 180,E1 -9011.998,E2 -9011.998} C_VEL
LIN {X 0,Y 439.465,Z 329.369,A -85,B 0,C 180,E1 -9015.775,E2 -9015.775} C_VEL
LIN {X 0,Y 439.443,Z 329.368,A -85,B 0,C 180,E1 -9019.336,E2 -9019.336} C_VEL
LIN {X 0,Y 439.367,Z 329.377,A -85,B 0,C 180,E1 -9022.575,E2 -9022.575} C_VEL
LIN {X 0,Y 439.382,Z 329.38,A -85,B 0,C 180,E1 -9025.586,E2 -9025.586} C_VEL
LIN {X 0,Y 439.416,Z 329.371,A -85,B 0,C 180,E1 -9028.673,E2 -9028.673} C_VEL
LIN {X 0,Y 439.373,Z 329.379,A -85,B 0,C 180,E1 -9032.03,E2 -9032.03} C_VEL
LIN {X 0,Y 439.397,Z 329.379,A -85,B 0,C 180,E1 -9035.34,E2 -9035.34} C_VEL
LIN {X 0,Y 439.392,Z 329.374,A -85,B 0,C 180,E1 -9038.594,E2 -9038.594} C_VEL
LIN {X 0,Y 439.39,Z 329.379,A -85,B 0,C 180,E1 -9041.257,E2 -9041.257} C_VEL
LIN {X 0,Y 439.401,Z 329.374,A -85,B 0,C 180,E1 -9044.729,E2 -9044.729} C_VEL
LIN {X 0,Y 439.397,Z 329.377,A -85,B 0,C 180,E1 -9047.795,E2 -9047.795} C_VEL
LIN {X 0,Y 439.427,Z 329.373,A -85,B 0,C 180,E1 -9050.227,E2 -9050.227} C_VEL
LIN {X 0,Y 439.378,Z 329.385,A -85,B 0,C 180,E1 -9053.713,E2 -9053.713} C_VEL
LIN {X 0,Y 439.374,Z 329.384,A -85,B 0,C 180,E1 -9057.054,E2 -9057.054} C_VEL
LIN {X 0,Y 439.425,Z 329.375,A -85,B 0,C 180,E1 -9060.803,E2 -9060.803} C_VEL
LIN {X 0,Y 439.496,Z 329.56,A -85,B 0,C 180,E1 -9061.201,E2 -9061.201} C_VEL
LIN {X 0,Y 442.792,Z 344.829,A -85,B 0,C 180,E1 -9064.12,E2 -9064.12} C_VEL
LIN {X 0,Y 443.158,Z 348.683,A -85,B 0,C 180,E1 -9064.816,E2 -9064.816} C_VEL
LIN {X 0,Y 441.936,Z 368.393,A -85,B 0,C 180,E1 -9068.178,E2 -9068.178} C_VEL
LIN {X 0,Y 446.438,Z 394.467,A -85,B 0,C 180,E1 -9068.835,E2 -9068.835} C_VEL
LIN {X 0,Y 445.039,Z 506.369,A -85,B 0,C 180,E1 -9070.662,E2 -9070.662} C_VEL
LIN {X 0,Y 444.581,Z 521.112,A -85,B 0,C 180,E1 -9071.091,E2 -9071.091} C_VEL
LIN {X 0,Y 443.924,Z 535,A -85,B 0,C 180,E1 -9071.682,E2 -9071.682} C_VEL
LIN {X 0,Y 443.183,Z 548.64,A -85,B 0,C 180,E1 -9072.464,E2 -9072.464} C_VEL
LIN {X 0,Y 442.304,Z 561.197,A -85,B 0,C 180,E1 -9073.381,E2 -9073.381} C_VEL
LIN {X 0,Y 441.406,Z 573.846,A -85,B 0,C 180,E1 -9074.532,E2 -9074.532} C_VEL
LIN {X 0,Y 440.678,Z 584.183,A -85,B 0,C 180,E1 -9075.688,E2 -9075.688} C_VEL
LIN {X 0,Y 440.027,Z 594.453,A -85,B 0,C 180,E1 -9077.079,E2 -9077.079} C_VEL
LIN {X 0,Y 439.477,Z 602.959,A -85,B 0,C 180,E1 -9078.469,E2 -9078.469} C_VEL
LIN {X 0,Y 438.919,Z 611.073,A -85,B 0,C 180,E1 -9080.088,E2 -9080.088} C_VEL
LIN {X 0,Y 438.606,Z 617.614,A -85,B 0,C 180,E1 -9081.708,E2 -9081.708} C_VEL
LIN {X 0,Y 438.447,Z 623.411,A -85,B 0,C 180,E1 -9083.558,E2 -9083.558} C_VEL
LIN {X 0,Y 438.319,Z 627.623,A -85,B 0,C 180,E1 -9085.402,E2 -9085.402} C_VEL
LIN {X 0,Y 438.336,Z 630.389,A -85,B 0,C 180,E1 -9087.243,E2 -9087.243} C_VEL
LIN {X 0,Y 438.25,Z 631.78,A -85,B 0,C 180,E1 -9089.081,E2 -9089.081} C_VEL
LIN {X 0,Y 438.25,Z 631.833,A -85,B 0,C 180,E1 -9090.919,E2 -9090.919} C_VEL
LIN {X 0,Y 438.336,Z 630.55,A -85,B 0,C 180,E1 -9092.757,E2 -9092.757} C_VEL
LIN {X 0,Y 438.319,Z 627.893,A -85,B 0,C 180,E1 -9094.598,E2 -9094.598} C_VEL
LIN {X 0,Y 438.446,Z 623.8,A -85,B 0,C 180,E1 -9096.443,E2 -9096.443} C_VEL
LIN {X 0,Y 438.623,Z 618.153,A -85,B 0,C 180,E1 -9098.291,E2 -9098.291} C_VEL
LIN {X 0,Y 438.955,Z 611.797,A -85,B 0,C 180,E1 -9099.911,E2 -9099.911} C_VEL
LIN {X 0,Y 439.517,Z 603.904,A -85,B 0,C 180,E1 -9101.53,E2 -9101.53} C_VEL
LIN {X 0,Y 440.085,Z 594.795,A -85,B 0,C 180,E1 -9103.057,E2 -9103.057} C_VEL
LIN {X 0,Y 440.789,Z 585.762,A -85,B 0,C 180,E1 -9104.308,E2 -9104.308} C_VEL
LIN {X 0,Y 441.627,Z 574.769,A -85,B 0,C 180,E1 -9105.578,E2 -9105.578} C_VEL
LIN {X 0,Y 442.707,Z 562.548,A -85,B 0,C 180,E1 -9106.723,E2 -9106.723} C_VEL
LIN {X 0,Y 443.523,Z 551.055,A -85,B 0,C 180,E1 -9107.6,E2 -9107.6} C_VEL
LIN {X 0,Y 444.241,Z 538.683,A -85,B 0,C 180,E1 -9108.359,E2 -9108.359} C_VEL
LIN {X 0,Y 444.928,Z 524.648,A -85,B 0,C 180,E1 -9109.014,E2 -9109.014} C_VEL
LIN {X 0,Y 445.565,Z 510.755,A -85,B 0,C 180,E1 -9109.464,E2 -9109.464} C_VEL
LIN {X 0,Y 445.916,Z 493.353,A -85,B 0,C 180,E1 -9109.807,E2 -9109.807} C_VEL
LIN {X 0,Y 447.102,Z 393.727,A -85,B 0,C 180,E1 -9111.44,E2 -9111.44} C_VEL
LIN {X 0,Y 443.099,Z 372.202,A -85,B 0,C 180,E1 -9112.029,E2 -9112.029} C_VEL
LIN {X 0,Y 442.296,Z 368.3,A -85,B 0,C 180,E1 -9112.148,E2 -9112.148} C_VEL
LIN {X 0,Y 443.403,Z 352.798,A -85,B 0,C 180,E1 -9114.837,E2 -9114.837} C_VEL
LIN {X 0,Y 443.66,Z 348.608,A -85,B 0,C 180,E1 -9115.573,E2 -9115.573} C_VEL
LIN {X 0,Y 441.344,Z 337.426,A -85,B 0,C 180,E1 -9117.761,E2 -9117.761} C_VEL
LIN {X 0,Y 439.446,Z 329.369,A -85,B 0,C 180,E1 -9119.425,E2 -9119.425} C_VEL
LIN {X 0,Y 439.374,Z 329.38,A -85,B 0,C 180,E1 -9122.946,E2 -9122.946} C_VEL
LIN {X 0,Y 439.375,Z 329.381,A -85,B 0,C 180,E1 -9126.287,E2 -9126.287} C_VEL
LIN {X 0,Y 439.403,Z 329.373,A -85,B 0,C 180,E1 -9129.849,E2 -9129.849} C_VEL
LIN {X 0,Y 439.382,Z 329.38,A -85,B 0,C 180,E1 -9132.627,E2 -9132.627} C_VEL
LIN {X 0,Y 439.401,Z 329.372,A -85,B 0,C 180,E1 -9135.271,E2 -9135.271} C_VEL
LIN {X 0,Y 439.391,Z 329.378,A -85,B 0,C 180,E1 -9138.744,E2 -9138.744} C_VEL
LIN {X 0,Y 439.378,Z 329.375,A -85,B 0,C 180,E1 -9141.608,E2 -9141.608} C_VEL
LIN {X 0,Y 439.4,Z 329.375,A -85,B 0,C 180,E1 -9144.844,E2 -9144.844} C_VEL
LIN {X 0,Y 439.376,Z 329.38,A -85,B 0,C 180,E1 -9148.14,E2 -9148.14} C_VEL
LIN {X 0,Y 439.411,Z 329.372,A -85,B 0,C 180,E1 -9151.604,E2 -9151.604} C_VEL
LIN {X 0,Y 439.383,Z 329.378,A -85,B 0,C 180,E1 -9154.414,E2 -9154.414} C_VEL
LIN {X 0,Y 439.367,Z 329.375,A -85,B 0,C 180,E1 -9157.425,E2 -9157.425} C_VEL
LIN {X 0,Y 439.444,Z 329.368,A -85,B 0,C 180,E1 -9160.664,E2 -9160.664} C_VEL
LIN {X 0,Y 439.466,Z 329.371,A -85,B 0,C 180,E1 -9164.225,E2 -9164.225} C_VEL
LIN {X 0,Y 439.487,Z 329.364,A -85,B 0,C 180,E1 -9168.002,E2 -9168.002} C_VEL
LIN {X 0,Y 439.506,Z 329.359,A -85,B 0,C 180,E1 -9171.726,E2 -9171.726} C_VEL
LIN {X 0,Y 439.608,Z 329.348,A -85,B 0,C 180,E1 -9174.496,E2 -9174.496} C_VEL
LIN {X 0,Y 439.63,Z 329.349,A -85,B 0,C 180,E1 -9178.168,E2 -9178.168} C_VEL
LIN {X 0,Y 439.692,Z 329.34,A -85,B 0,C 180,E1 -9180,E2 -9180} C_VEL
LIN {X 0,Y 439.632,Z 329.342,A -85,B 0,C 180,E1 -9182.749,E2 -9182.749} C_VEL
LIN {X 0,Y 439.562,Z 329.347,A -85,B 0,C 180,E1 -9186.426,E2 -9186.426} C_VEL
LIN {X 0,Y 439.494,Z 329.363,A -85,B 0,C 180,E1 -9189.202,E2 -9189.202} C_VEL
LIN {X 0,Y 439.469,Z 329.362,A -85,B 0,C 180,E1 -9192.938,E2 -9192.938} C_VEL
LIN {X 0,Y 439.401,Z 329.369,A -85,B 0,C 180,E1 -9196.326,E2 -9196.326} C_VEL
LIN {X 0,Y 439.381,Z 329.379,A -85,B 0,C 180,E1 -9199.628,E2 -9199.628} C_VEL
LIN {X 0,Y 439.363,Z 329.378,A -85,B 0,C 180,E1 -9202.576,E2 -9202.576} C_VEL
LIN {X 0,Y 439.37,Z 329.379,A -85,B 0,C 180,E1 -9205.587,E2 -9205.587} C_VEL
LIN {X 0,Y 439.38,Z 329.372,A -85,B 0,C 180,E1 -9208.677,E2 -9208.677} C_VEL
LIN {X 0,Y 439.355,Z 329.379,A -85,B 0,C 180,E1 -9212.026,E2 -9212.026} C_VEL
LIN {X 0,Y 439.39,Z 329.372,A -85,B 0,C 180,E1 -9215.339,E2 -9215.339} C_VEL
LIN {X 0,Y 439.351,Z 329.379,A -85,B 0,C 180,E1 -9218.599,E2 -9218.599} C_VEL
LIN {X 0,Y 439.348,Z 329.38,A -85,B 0,C 180,E1 -9222.211,E2 -9222.211} C_VEL
LIN {X 0,Y 439.377,Z 329.376,A -85,B 0,C 180,E1 -9225.267,E2 -9225.267} C_VEL
LIN {X 0,Y 439.361,Z 329.383,A -85,B 0,C 180,E1 -9228.748,E2 -9228.748} C_VEL
LIN {X 0,Y 439.353,Z 329.385,A -85,B 0,C 180,E1 -9231.612,E2 -9231.612} C_VEL
LIN {X 0,Y 439.39,Z 329.38,A -85,B 0,C 180,E1 -9234.843,E2 -9234.843} C_VEL
LIN {X 0,Y 439.348,Z 329.381,A -85,B 0,C 180,E1 -9238.137,E2 -9238.137} C_VEL
LIN {X 0,Y 439.406,Z 329.579,A -85,B 0,C 180,E1 -9239.287,E2 -9239.287} C_VEL
LIN {X 0,Y 442.027,Z 341.792,A -85,B 0,C 180,E1 -9242.028,E2 -9242.028} C_VEL
LIN {X 0,Y 442.611,Z 346.139,A -85,B 0,C 180,E1 -9242.931,E2 -9242.931} C_VEL
LIN {X 0,Y 447.401,Z 366.97,A -85,B 0,C 180,E1 -9243.559,E2 -9243.559} C_VEL
LIN {X 0,Y 446.023,Z 482.374,A -85,B 0,C 180,E1 -9245.474,E2 -9245.474} C_VEL
LIN {X 0,Y 445.551,Z 496.717,A -85,B 0,C 180,E1 -9245.89,E2 -9245.89} C_VEL
LIN {X 0,Y 444.817,Z 510.559,A -85,B 0,C 180,E1 -9246.476,E2 -9246.476} C_VEL
LIN {X 0,Y 444.177,Z 523.106,A -85,B 0,C 180,E1 -9247.191,E2 -9247.191} C_VEL
LIN {X 0,Y 443.972,Z 526.434,A -85,B 0,C 180,E1 -9247.409,E2 -9247.409} C_VEL
LIN {X 0,Y 443.079,Z 531.648,A -85,B 0,C 180,E1 -9247.746,E2 -9247.746} C_VEL
LIN {X 0,Y 439.786,Z 539.968,A -85,B 0,C 180,E1 -9248.298,E2 -9248.298} C_VEL
LIN {X 0,Y 436.364,Z 547.92,A -85,B 0,C 180,E1 -9248.93,E2 -9248.93} C_VEL
LIN {X 0,Y 435.28,Z 552.537,A -85,B 0,C 180,E1 -9249.39,E2 -9249.39} C_VEL
LIN {X 0,Y 434.371,Z 562.801,A -85,B 0,C 180,E1 -9250.629,E2 -9250.629} C_VEL
LIN {X 0,Y 433.526,Z 572.589,A -85,B 0,C 180,E1 -9252.06,E2 -9252.06} C_VEL
LIN {X 0,Y 432.811,Z 581.315,A -85,B 0,C 180,E1 -9253.616,E2 -9253.616} C_VEL
LIN {X 0,Y 432.246,Z 588.396,A -85,B 0,C 180,E1 -9255.162,E2 -9255.162} C_VEL
LIN {X 0,Y 431.833,Z 594.556,A -85,B 0,C 180,E1 -9256.83,E2 -9256.83} C_VEL
LIN {X 0,Y 431.474,Z 599.969,A -85,B 0,C 180,E1 -9258.728,E2 -9258.728} C_VEL
LIN {X 0,Y 431.271,Z 603.783,A -85,B 0,C 180,E1 -9260.621,E2 -9260.621} C_VEL
LIN {X 0,Y 431.216,Z 606.173,A -85,B 0,C 180,E1 -9262.508,E2 -9262.508} C_VEL
LIN {X 0,Y 431.21,Z 607.216,A -85,B 0,C 180,E1 -9264.388,E2 -9264.388} C_VEL
LIN {X 0,Y 431.164,Z 606.941,A -85,B 0,C 180,E1 -9266.262,E2 -9266.262} C_VEL
LIN {X 0,Y 431.27,Z 606.306,A -85,B 0,C 180,E1 -9267.198,E2 -9267.198} C_VEL
LIN {X 0,Y 431.202,Z 604.05,A -85,B 0,C 180,E1 -9269.066,E2 -9269.066} C_VEL
LIN {X 0,Y 431.332,Z 600.412,A -85,B 0,C 180,E1 -9270.934,E2 -9270.934} C_VEL
LIN {X 0,Y 431.601,Z 595.289,A -85,B 0,C 180,E1 -9272.8,E2 -9272.8} C_VEL
LIN {X 0,Y 432.095,Z 590.309,A -85,B 0,C 180,E1 -9274.197,E2 -9274.197} C_VEL
LIN {X 0,Y 432.568,Z 583.217,A -85,B 0,C 180,E1 -9275.828,E2 -9275.828} C_VEL
LIN {X 0,Y 433.158,Z 574.468,A -85,B 0,C 180,E1 -9277.458,E2 -9277.458} C_VEL
LIN {X 0,Y 433.785,Z 565.628,A -85,B 0,C 180,E1 -9278.807,E2 -9278.807} C_VEL
LIN {X 0,Y 434.677,Z 555.169,A -85,B 0,C 180,E1 -9280.127,E2 -9280.127} C_VEL
LIN {X 0,Y 435.413,Z 544.031,A -85,B 0,C 180,E1 -9281.286,E2 -9281.286} C_VEL
LIN {X 0,Y 436.272,Z 531.719,A -85,B 0,C 180,E1 -9282.325,E2 -9282.325} C_VEL
LIN {X 0,Y 437.015,Z 519.868,A -85,B 0,C 180,E1 -9283.13,E2 -9283.13} C_VEL
LIN {X 0,Y 437.721,Z 506.901,A -85,B 0,C 180,E1 -9283.818,E2 -9283.818} C_VEL
LIN {X 0,Y 438.217,Z 492.947,A -85,B 0,C 180,E1 -9284.364,E2 -9284.364} C_VEL
LIN {X 0,Y 438.576,Z 478.262,A -85,B 0,C 180,E1 -9284.738,E2 -9284.738} C_VEL
LIN {X 0,Y 439.935,Z 367.654,A -85,B 0,C 180,E1 -9286.561,E2 -9286.561} C_VEL
LIN {X 0,Y 435.295,Z 346.013,A -85,B 0,C 180,E1 -9287.174,E2 -9287.174} C_VEL
LIN {X 0,Y 434.432,Z 340.282,A -85,B 0,C 180,E1 -9288.389,E2 -9288.389} C_VEL
LIN {X 0,Y 432.338,Z 330.26,A -85,B 0,C 180,E1 -9290.643,E2 -9290.643} C_VEL
LIN {X 0,Y 432.335,Z 330.257,A -85,B 0,C 180,E1 -9293.979,E2 -9293.979} C_VEL
LIN {X 0,Y 432.292,Z 330.266,A -85,B 0,C 180,E1 -9297.079,E2 -9297.079} C_VEL
LIN {X 0,Y 432.331,Z 330.253,A -85,B 0,C 180,E1 -9300.261,E2 -9300.261} C_VEL
LIN {X 0,Y 432.31,Z 330.258,A -85,B 0,C 180,E1 -9303.555,E2 -9303.555} C_VEL
LIN {X 0,Y 432.333,Z 330.254,A -85,B 0,C 180,E1 -9305.818,E2 -9305.818} C_VEL
LIN {X 0,Y 432.314,Z 330.261,A -85,B 0,C 180,E1 -9308.709,E2 -9308.709} C_VEL
LIN {X 0,Y 432.303,Z 330.256,A -85,B 0,C 180,E1 -9311.801,E2 -9311.801} C_VEL
LIN {X 0,Y 432.335,Z 330.257,A -85,B 0,C 180,E1 -9314.348,E2 -9314.348} C_VEL
LIN {X 0,Y 432.303,Z 330.259,A -85,B 0,C 180,E1 -9317.019,E2 -9317.019} C_VEL
LIN {X 0,Y 432.29,Z 330.258,A -85,B 0,C 180,E1 -9319.828,E2 -9319.828} C_VEL
LIN {X 0,Y 432.297,Z 330.258,A -85,B 0,C 180,E1 -9323.021,E2 -9323.021} C_VEL
LIN {X 0,Y 432.335,Z 330.255,A -85,B 0,C 180,E1 -9326.002,E2 -9326.002} C_VEL
LIN {X 0,Y 432.334,Z 330.253,A -85,B 0,C 180,E1 -9329.493,E2 -9329.493} C_VEL
LIN {X 0,Y 432.318,Z 330.254,A -85,B 0,C 180,E1 -9331.872,E2 -9331.872} C_VEL
LIN {X 0,Y 432.327,Z 330.255,A -85,B 0,C 180,E1 -9334.997,E2 -9334.997} C_VEL
LIN {X 0,Y 432.358,Z 330.249,A -85,B 0,C 180,E1 -9338.045,E2 -9338.045} C_VEL
LIN {X 0,Y 432.384,Z 330.24,A -85,B 0,C 180,E1 -9341.029,E2 -9341.029} C_VEL
LIN {X 0,Y 432.389,Z 330.249,A -85,B 0,C 180,E1 -9343.959,E2 -9343.959} C_VEL
LIN {X 0,Y 432.463,Z 330.231,A -85,B 0,C 180,E1 -9347.803,E2 -9347.803} C_VEL
LIN {X 0,Y 432.467,Z 330.231,A -85,B 0,C 180,E1 -9351.59,E2 -9351.59} C_VEL
LIN {X 0,Y 432.576,Z 330.226,A -85,B 0,C 180,E1 -9354.406,E2 -9354.406} C_VEL
LIN {X 0,Y 432.605,Z 330.226,A -85,B 0,C 180,E1 -9358.138,E2 -9358.138} C_VEL
LIN {X 0,Y 432.55,Z 330.222,A -85,B 0,C 180,E1 -9360.931,E2 -9360.931} C_VEL
LIN {X 0,Y 432.564,Z 330.225,A -85,B 0,C 180,E1 -9362.794,E2 -9362.794} C_VEL
LIN {X 0,Y 432.581,Z 330.222,A -85,B 0,C 180,E1 -9365.594,E2 -9365.594} C_VEL
LIN {X 0,Y 432.466,Z 330.238,A -85,B 0,C 180,E1 -9368.41,E2 -9368.41} C_VEL
LIN {X 0,Y 432.462,Z 330.241,A -85,B 0,C 180,E1 -9372.196,E2 -9372.196} C_VEL
LIN {X 0,Y 432.433,Z 330.246,A -85,B 0,C 180,E1 -9376.039,E2 -9376.039} C_VEL
LIN {X 0,Y 432.389,Z 330.248,A -85,B 0,C 180,E1 -9379.485,E2 -9379.485} C_VEL
LIN {X 0,Y 432.32,Z 330.254,A -85,B 0,C 180,E1 -9382.964,E2 -9382.964} C_VEL
LIN {X 0,Y 432.341,Z 330.253,A -85,B 0,C 180,E1 -9385.002,E2 -9385.002} C_VEL
LIN {X 0,Y 432.38,Z 330.25,A -85,B 0,C 180,E1 -9388.123,E2 -9388.123} C_VEL
LIN {X 0,Y 432.323,Z 330.259,A -85,B 0,C 180,E1 -9391.346,E2 -9391.346} C_VEL
LIN {X 0,Y 432.342,Z 330.254,A -85,B 0,C 180,E1 -9394.677,E2 -9394.677} C_VEL
LIN {X 0,Y 432.349,Z 330.253,A -85,B 0,C 180,E1 -9398.149,E2 -9398.149} C_VEL
LIN {X 0,Y 432.335,Z 330.261,A -85,B 0,C 180,E1 -9401.602,E2 -9401.602} C_VEL
LIN {X 0,Y 432.335,Z 330.255,A -85,B 0,C 180,E1 -9404.347,E2 -9404.347} C_VEL
LIN {X 0,Y 432.321,Z 330.257,A -85,B 0,C 180,E1 -9407.015,E2 -9407.015} C_VEL
LIN {X 0,Y 432.334,Z 330.258,A -85,B 0,C 180,E1 -9409.821,E2 -9409.821} C_VEL
LIN {X 0,Y 432.317,Z 330.263,A -85,B 0,C 180,E1 -9413.023,E2 -9413.023} C_VEL
LIN {X 0,Y 432.361,Z 330.256,A -85,B 0,C 180,E1 -9415.996,E2 -9415.996} C_VEL
LIN {X 0,Y 432.349,Z 330.258,A -85,B 0,C 180,E1 -9419.489,E2 -9419.489} C_VEL
LIN {X 0,Y 432.405,Z 330.291,A -85,B 0,C 180,E1 -9420.89,E2 -9420.89} C_VEL
LIN {X 0,Y 435.486,Z 344.443,A -85,B 0,C 180,E1 -9423.653,E2 -9423.653} C_VEL
LIN {X 0,Y 436.283,Z 349.487,A -85,B 0,C 180,E1 -9424.598,E2 -9424.598} C_VEL
LIN {X 0,Y 435.046,Z 368.237,A -85,B 0,C 180,E1 -9427.85,E2 -9427.85} C_VEL
LIN {X 0,Y 439.752,Z 396.01,A -85,B 0,C 180,E1 -9428.553,E2 -9428.553} C_VEL
LIN {X 0,Y 438.276,Z 506.365,A -85,B 0,C 180,E1 -9430.382,E2 -9430.382} C_VEL
LIN {X 0,Y 437.793,Z 521.039,A -85,B 0,C 180,E1 -9430.817,E2 -9430.817} C_VEL
LIN {X 0,Y 437.132,Z 534.719,A -85,B 0,C 180,E1 -9431.408,E2 -9431.408} C_VEL
LIN {X 0,Y 436.364,Z 548.074,A -85,B 0,C 180,E1 -9432.181,E2 -9432.181} C_VEL
LIN {X 0,Y 435.481,Z 560.705,A -85,B 0,C 180,E1 -9433.112,E2 -9433.112} C_VEL
LIN {X 0,Y 434.619,Z 572.227,A -85,B 0,C 180,E1 -9434.164,E2 -9434.164} C_VEL
LIN {X 0,Y 433.895,Z 581.82,A -85,B 0,C 180,E1 -9435.22,E2 -9435.22} C_VEL
LIN {X 0,Y 433.223,Z 590.849,A -85,B 0,C 180,E1 -9436.395,E2 -9436.395} C_VEL
LIN {X 0,Y 432.588,Z 599.928,A -85,B 0,C 180,E1 -9437.807,E2 -9437.807} C_VEL
LIN {X 0,Y 432.025,Z 608.609,A -85,B 0,C 180,E1 -9439.455,E2 -9439.455} C_VEL
LIN {X 0,Y 431.617,Z 615.608,A -85,B 0,C 180,E1 -9441.101,E2 -9441.101} C_VEL
LIN {X 0,Y 431.407,Z 621.886,A -85,B 0,C 180,E1 -9442.982,E2 -9442.982} C_VEL
LIN {X 0,Y 431.278,Z 625.454,A -85,B 0,C 180,E1 -9444.389,E2 -9444.389} C_VEL
LIN {X 0,Y 431.177,Z 628.944,A -85,B 0,C 180,E1 -9446.262,E2 -9446.262} C_VEL
LIN {X 0,Y 431.2,Z 631.033,A -85,B 0,C 180,E1 -9448.132,E2 -9448.132} C_VEL
LIN {X 0,Y 431.165,Z 631.769,A -85,B 0,C 180,E1 -9450,E2 -9450} C_VEL
LIN {X 0,Y 431.2,Z 631.171,A -85,B 0,C 180,E1 -9451.868,E2 -9451.868} C_VEL
LIN {X 0,Y 431.176,Z 629.225,A -85,B 0,C 180,E1 -9453.738,E2 -9453.738} C_VEL
LIN {X 0,Y 431.278,Z 625.879,A -85,B 0,C 180,E1 -9455.611,E2 -9455.611} C_VEL
LIN {X 0,Y 431.391,Z 622.404,A -85,B 0,C 180,E1 -9457.018,E2 -9457.018} C_VEL
LIN {X 0,Y 431.648,Z 616.395,A -85,B 0,C 180,E1 -9458.898,E2 -9458.898} C_VEL
LIN {X 0,Y 432.048,Z 609.642,A -85,B 0,C 180,E1 -9460.545,E2 -9460.545} C_VEL
LIN {X 0,Y 432.721,Z 601.258,A -85,B 0,C 180,E1 -9462.189,E2 -9462.189} C_VEL
LIN {X 0,Y 433.299,Z 592.862,A -85,B 0,C 180,E1 -9463.555,E2 -9463.555} C_VEL
LIN {X 0,Y 434.174,Z 581.986,A -85,B 0,C 180,E1 -9465.01,E2 -9465.01} C_VEL
LIN {X 0,Y 435.206,Z 570.191,A -85,B 0,C 180,E1 -9466.295,E2 -9466.295} C_VEL
LIN {X 0,Y 436.18,Z 558.372,A -85,B 0,C 180,E1 -9467.343,E2 -9467.343} C_VEL
LIN {X 0,Y 437.166,Z 544.609,A -85,B 0,C 180,E1 -9468.318,E2 -9468.318} C_VEL
LIN {X 0,Y 437.986,Z 530.353,A -85,B 0,C 180,E1 -9469.083,E2 -9469.083} C_VEL
LIN {X 0,Y 438.666,Z 517.171,A -85,B 0,C 180,E1 -9469.6,E2 -9469.6} C_VEL
LIN {X 0,Y 439.174,Z 502.871,A -85,B 0,C 180,E1 -9469.972,E2 -9469.972} C_VEL
LIN {X 0,Y 440.58,Z 394.789,A -85,B 0,C 180,E1 -9471.778,E2 -9471.778} C_VEL
LIN {X 0,Y 436.502,Z 372.94,A -85,B 0,C 180,E1 -9472.392,E2 -9472.392} C_VEL
LIN {X 0,Y 435.463,Z 368.092,A -85,B 0,C 180,E1 -9472.544,E2 -9472.544} C_VEL
LIN {X 0,Y 436.65,Z 352.881,A -85,B 0,C 180,E1 -9475.228,E2 -9475.228} C_VEL
LIN {X 0,Y 436.758,Z 349.979,A -85,B 0,C 180,E1 -9475.751,E2 -9475.751} C_VEL
LIN {X 0,Y 434.438,Z 338.813,A -85,B 0,C 180,E1 -9477.979,E2 -9477.979} C_VEL
LIN {X 0,Y 432.374,Z 330.251,A -85,B 0,C 180,E1 -9479.787,E2 -9479.787} C_VEL
LIN {X 0,Y 432.341,Z 330.253,A -85,B 0,C 180,E1 -9483.552,E2 -9483.552} C_VEL
LIN {X 0,Y 432.339,Z 330.256,A -85,B 0,C 180,E1 -9485.818,E2 -9485.818} C_VEL
LIN {X 0,Y 432.339,Z 330.253,A -85,B 0,C 180,E1 -9489.344,E2 -9489.344} C_VEL
LIN {X 0,Y 432.335,Z 330.254,A -85,B 0,C 180,E1 -9491.797,E2 -9491.797} C_VEL
LIN {X 0,Y 432.335,Z 330.258,A -85,B 0,C 180,E1 -9494.348,E2 -9494.348} C_VEL
LIN {X 0,Y 432.322,Z 330.256,A -85,B 0,C 180,E1 -9497.016,E2 -9497.016} C_VEL
LIN {X 0,Y 432.343,Z 330.254,A -85,B 0,C 180,E1 -9499.82,E2 -9499.82} C_VEL
LIN {X 0,Y 432.307,Z 330.255,A -85,B 0,C 180,E1 -9503.022,E2 -9503.022} C_VEL
LIN {X 0,Y 432.361,Z 330.254,A -85,B 0,C 180,E1 -9505.997,E2 -9505.997} C_VEL
LIN {X 0,Y 432.349,Z 330.251,A -85,B 0,C 180,E1 -9509.49,E2 -9509.49} C_VEL
LIN {X 0,Y 432.35,Z 330.254,A -85,B 0,C 180,E1 -9511.875,E2 -9511.875} C_VEL
LIN {X 0,Y 432.382,Z 330.248,A -85,B 0,C 180,E1 -9515.539,E2 -9515.539} C_VEL
LIN {X 0,Y 432.353,Z 330.25,A -85,B 0,C 180,E1 -9519.046,E2 -9519.046} C_VEL
LIN {X 0,Y 432.376,Z 330.248,A -85,B 0,C 180,E1 -9522.011,E2 -9522.011} C_VEL
LIN {X 0,Y 432.398,Z 330.245,A -85,B 0,C 180,E1 -9524.927,E2 -9524.927} C_VEL
LIN {X 0,Y 432.463,Z 330.236,A -85,B 0,C 180,E1 -9527.804,E2 -9527.804} C_VEL
LIN {X 0,Y 432.467,Z 330.235,A -85,B 0,C 180,E1 -9531.59,E2 -9531.59} C_VEL
LIN {X 0,Y 432.581,Z 330.224,A -85,B 0,C 180,E1 -9534.406,E2 -9534.406} C_VEL
LIN {X 0,Y 432.6,Z 330.225,A -85,B 0,C 180,E1 -9538.138,E2 -9538.138} C_VEL
LIN {X 0,Y 432.643,Z 330.218,A -85,B 0,C 180,E1 -9540,E2 -9540} C_VEL
LIN {X 0,Y 432.584,Z 330.219,A -85,B 0,C 180,E1 -9542.794,E2 -9542.794} C_VEL
LIN {X 0,Y 432.574,Z 330.228,A -85,B 0,C 180,E1 -9545.594,E2 -9545.594} C_VEL
LIN {X 0,Y 432.466,Z 330.238,A -85,B 0,C 180,E1 -9548.41,E2 -9548.41} C_VEL
LIN {X 0,Y 432.463,Z 330.237,A -85,B 0,C 180,E1 -9552.197,E2 -9552.197} C_VEL
LIN {X 0,Y 432.389,Z 330.244,A -85,B 0,C 180,E1 -9556.041,E2 -9556.041} C_VEL
LIN {X 0,Y 432.351,Z 330.257,A -85,B 0,C 180,E1 -9559.47,E2 -9559.47} C_VEL
LIN {X 0,Y 432.344,Z 330.254,A -85,B 0,C 180,E1 -9562.093,E2 -9562.093} C_VEL
LIN {X 0,Y 432.326,Z 330.252,A -85,B 0,C 180,E1 -9565.003,E2 -9565.003} C_VEL
LIN {X 0,Y 432.318,Z 330.252,A -85,B 0,C 180,E1 -9568.128,E2 -9568.128} C_VEL
LIN {X 0,Y 432.307,Z 330.246,A -85,B 0,C 180,E1 -9571.348,E2 -9571.348} C_VEL
LIN {X 0,Y 432.328,Z 330.254,A -85,B 0,C 180,E1 -9574.679,E2 -9574.679} C_VEL
LIN {X 0,Y 432.321,Z 330.255,A -85,B 0,C 180,E1 -9578.152,E2 -9578.152} C_VEL
LIN {X 0,Y 432.303,Z 330.26,A -85,B 0,C 180,E1 -9581.801,E2 -9581.801} C_VEL
LIN {X 0,Y 432.335,Z 330.255,A -85,B 0,C 180,E1 -9584.348,E2 -9584.348} C_VEL
LIN {X 0,Y 432.303,Z 330.26,A -85,B 0,C 180,E1 -9587.019,E2 -9587.019} C_VEL
LIN {X 0,Y 432.29,Z 330.262,A -85,B 0,C 180,E1 -9589.828,E2 -9589.828} C_VEL
LIN {X 0,Y 432.296,Z 330.264,A -85,B 0,C 180,E1 -9593.021,E2 -9593.021} C_VEL
LIN {X 0,Y 432.333,Z 330.255,A -85,B 0,C 180,E1 -9596.003,E2 -9596.003} C_VEL
LIN {X 0,Y 432.328,Z 330.357,A -85,B 0,C 180,E1 -9598.926,E2 -9598.926} C_VEL
LIN {X 0,Y 435.051,Z 342.934,A -85,B 0,C 180,E1 -9601.802,E2 -9601.802} C_VEL
LIN {X 0,Y 435.669,Z 346.346,A -85,B 0,C 180,E1 -9602.529,E2 -9602.529} C_VEL
LIN {X 0,Y 439.643,Z 362.213,A -85,B 0,C 180,E1 -9603.041,E2 -9603.041} C_VEL
LIN {X 0,Y 440.936,Z 368.706,A -85,B 0,C 180,E1 -9603.228,E2 -9603.228} C_VEL
LIN {X 0,Y 439.418,Z 482.661,A -85,B 0,C 180,E1 -9605.144,E2 -9605.144} C_VEL
LIN {X 0,Y 438.921,Z 497.105,A -85,B 0,C 180,E1 -9605.571,E2 -9605.571} C_VEL
LIN {X 0,Y 438.207,Z 510.061,A -85,B 0,C 180,E1 -9606.121,E2 -9606.121} C_VEL
LIN {X 0,Y 437.554,Z 522.439,A -85,B 0,C 180,E1 -9606.826,E2 -9606.826} C_VEL
LIN {X 0,Y 436.578,Z 535.509,A -85,B 0,C 180,E1 -9607.771,E2 -9607.771} C_VEL
LIN {X 0,Y 435.655,Z 547.326,A -85,B 0,C 180,E1 -9608.841,E2 -9608.841} C_VEL
LIN {X 0,Y 435.28,Z 552.537,A -85,B 0,C 180,E1 -9609.39,E2 -9609.39} C_VEL
LIN {X 0,Y 434.201,Z 557.071,A -85,B 0,C 180,E1 -9609.876,E2 -9609.876} C_VEL
LIN {X 0,Y 430.772,Z 564.199,A -85,B 0,C 180,E1 -9610.669,E2 -9610.669} C_VEL
LIN {X 0,Y 427.416,Z 570.887,A -85,B 0,C 180,E1 -9611.535,E2 -9611.535} C_VEL
LIN {X 0,Y 426.463,Z 574.652,A -85,B 0,C 180,E1 -9612.13,E2 -9612.13} C_VEL
LIN {X 0,Y 425.752,Z 582.993,A -85,B 0,C 180,E1 -9613.702,E2 -9613.702} C_VEL
LIN {X 0,Y 425.18,Z 589.357,A -85,B 0,C 180,E1 -9615.155,E2 -9615.155} C_VEL
LIN {X 0,Y 424.82,Z 594.559,A -85,B 0,C 180,E1 -9616.608,E2 -9616.608} C_VEL
LIN {X 0,Y 424.409,Z 600.03,A -85,B 0,C 180,E1 -9618.538,E2 -9618.538} C_VEL
LIN {X 0,Y 424.19,Z 603.896,A -85,B 0,C 180,E1 -9620.463,E2 -9620.463} C_VEL
LIN {X 0,Y 424.12,Z 606.326,A -85,B 0,C 180,E1 -9622.382,E2 -9622.382} C_VEL
LIN {X 0,Y 424.125,Z 607.408,A -85,B 0,C 180,E1 -9624.294,E2 -9624.294} C_VEL
LIN {X 0,Y 424.074,Z 607.172,A -85,B 0,C 180,E1 -9626.199,E2 -9626.199} C_VEL
LIN {X 0,Y 424.165,Z 605.616,A -85,B 0,C 180,E1 -9628.101,E2 -9628.101} C_VEL
LIN {X 0,Y 424.163,Z 602.72,A -85,B 0,C 180,E1 -9630,E2 -9630} C_VEL
LIN {X 0,Y 424.338,Z 598.4,A -85,B 0,C 180,E1 -9631.898,E2 -9631.898} C_VEL
LIN {X 0,Y 424.791,Z 592.518,A -85,B 0,C 180,E1 -9633.795,E2 -9633.795} C_VEL
LIN {X 0,Y 425.337,Z 585.896,A -85,B 0,C 180,E1 -9635.452,E2 -9635.452} C_VEL
LIN {X 0,Y 425.861,Z 578.962,A -85,B 0,C 180,E1 -9636.872,E2 -9636.872} C_VEL
LIN {X 0,Y 426.414,Z 570.914,A -85,B 0,C 180,E1 -9638.251,E2 -9638.251} C_VEL
LIN {X 0,Y 427.317,Z 560.66,A -85,B 0,C 180,E1 -9639.705,E2 -9639.705} C_VEL
LIN {X 0,Y 428.207,Z 549.483,A -85,B 0,C 180,E1 -9640.999,E2 -9640.999} C_VEL
LIN {X 0,Y 429.04,Z 538.382,A -85,B 0,C 180,E1 -9642.055,E2 -9642.055} C_VEL
LIN {X 0,Y 429.889,Z 526.285,A -85,B 0,C 180,E1 -9642.991,E2 -9642.991} C_VEL
LIN {X 0,Y 430.585,Z 512.884,A -85,B 0,C 180,E1 -9643.81,E2 -9643.81} C_VEL
LIN {X 0,Y 431.301,Z 498.808,A -85,B 0,C 180,E1 -9644.449,E2 -9644.449} C_VEL
LIN {X 0,Y 431.725,Z 484.99,A -85,B 0,C 180,E1 -9644.886,E2 -9644.886} C_VEL
LIN {X 0,Y 432.074,Z 461.113,A -85,B 0,C 180,E1 -9645.327,E2 -9645.327} C_VEL
LIN {X 0,Y 433.29,Z 368.807,A -85,B 0,C 180,E1 -9646.864,E2 -9646.864} C_VEL
LIN {X 0,Y 428.314,Z 346.288,A -85,B 0,C 180,E1 -9647.509,E2 -9647.509} C_VEL
LIN {X 0,Y 426.186,Z 335.15,A -85,B 0,C 180,E1 -9649.955,E2 -9649.955} C_VEL
LIN {X 0,Y 425.318,Z 331.135,A -85,B 0,C 180,E1 -9650.873,E2 -9650.873} C_VEL
LIN {X 0,Y 425.296,Z 331.137,A -85,B 0,C 180,E1 -9654.649,E2 -9654.649} C_VEL
LIN {X 0,Y 425.24,Z 331.141,A -85,B 0,C 180,E1 -9657.566,E2 -9657.566} C_VEL
LIN {X 0,Y 425.287,Z 331.132,A -85,B 0,C 180,E1 -9660.759,E2 -9660.759} C_VEL
LIN {X 0,Y 425.29,Z 331.133,A -85,B 0,C 180,E1 -9664.283,E2 -9664.283} C_VEL
LIN {X 0,Y 425.27,Z 331.134,A -85,B 0,C 180,E1 -9667.695,E2 -9667.695} C_VEL
LIN {X 0,Y 425.247,Z 331.135,A -85,B 0,C 180,E1 -9671.382,E2 -9671.382} C_VEL
LIN {X 0,Y 425.286,Z 331.134,A -85,B 0,C 180,E1 -9674.716,E2 -9674.716} C_VEL
LIN {X 0,Y 425.265,Z 331.135,A -85,B 0,C 180,E1 -9678.046,E2 -9678.046} C_VEL
LIN {X 0,Y 425.267,Z 331.134,A -85,B 0,C 180,E1 -9681.097,E2 -9681.097} C_VEL
LIN {X 0,Y 425.295,Z 331.136,A -85,B 0,C 180,E1 -9684.663,E2 -9684.663} C_VEL
LIN {X 0,Y 425.255,Z 331.132,A -85,B 0,C 180,E1 -9688.072,E2 -9688.072} C_VEL
LIN {X 0,Y 425.295,Z 331.127,A -85,B 0,C 180,E1 -9691.365,E2 -9691.365} C_VEL
LIN {X 0,Y 425.263,Z 331.14,A -85,B 0,C 180,E1 -9694.552,E2 -9694.552} C_VEL
LIN {X 0,Y 425.294,Z 331.127,A -85,B 0,C 180,E1 -9697.73,E2 -9697.73} C_VEL
LIN {X 0,Y 425.363,Z 331.114,A -85,B 0,C 180,E1 -9700.704,E2 -9700.704} C_VEL
LIN {X 0,Y 425.322,Z 331.127,A -85,B 0,C 180,E1 -9703.685,E2 -9703.685} C_VEL
LIN {X 0,Y 425.397,Z 331.109,A -85,B 0,C 180,E1 -9707.096,E2 -9707.096} C_VEL
LIN {X 0,Y 425.4,Z 331.11,A -85,B 0,C 180,E1 -9710.49,E2 -9710.49} C_VEL
LIN {X 0,Y 425.481,Z 331.107,A -85,B 0,C 180,E1 -9713.36,E2 -9713.36} C_VEL
LIN {X 0,Y 425.357,Z 331.121,A -85,B 0,C 180,E1 -9715.261,E2 -9715.261} C_VEL
LIN {X 0,Y 425.574,Z 331.101,A -85,B 0,C 180,E1 -9718.107,E2 -9718.107} C_VEL
LIN {X 0,Y 425.513,Z 331.098,A -85,B 0,C 180,E1 -9720.946,E2 -9720.946} C_VEL
LIN {X 0,Y 425.519,Z 331.102,A -85,B 0,C 180,E1 -9722.84,E2 -9722.84} C_VEL
LIN {X 0,Y 425.535,Z 331.101,A -85,B 0,C 180,E1 -9725.687,E2 -9725.687} C_VEL
LIN {X 0,Y 425.41,Z 331.116,A -85,B 0,C 180,E1 -9728.55,E2 -9728.55} C_VEL
LIN {X 0,Y 425.415,Z 331.117,A -85,B 0,C 180,E1 -9732.401,E2 -9732.401} C_VEL
LIN {X 0,Y 425.391,Z 331.121,A -85,B 0,C 180,E1 -9736.311,E2 -9736.311} C_VEL
LIN {X 0,Y 425.331,Z 331.129,A -85,B 0,C 180,E1 -9739.635,E2 -9739.635} C_VEL
LIN {X 0,Y 425.307,Z 331.13,A -85,B 0,C 180,E1 -9743.365,E2 -9743.365} C_VEL
LIN {X 0,Y 425.307,Z 331.13,A -85,B 0,C 180,E1 -9746.498,E2 -9746.498} C_VEL
LIN {X 0,Y 425.291,Z 331.135,A -85,B 0,C 180,E1 -9749.719,E2 -9749.719} C_VEL
LIN {X 0,Y 425.284,Z 331.132,A -85,B 0,C 180,E1 -9753.048,E2 -9753.048} C_VEL
LIN {X 0,Y 425.286,Z 331.137,A -85,B 0,C 180,E1 -9755.929,E2 -9755.929} C_VEL
LIN {X 0,Y 425.305,Z 331.13,A -85,B 0,C 180,E1 -9759.044,E2 -9759.044} C_VEL
LIN {X 0,Y 425.276,Z 331.134,A -85,B 0,C 180,E1 -9762.653,E2 -9762.653} C_VEL
LIN {X 0,Y 425.262,Z 331.136,A -85,B 0,C 180,E1 -9766.044,E2 -9766.044} C_VEL
LIN {X 0,Y 425.275,Z 331.134,A -85,B 0,C 180,E1 -9768.621,E2 -9768.621} C_VEL
LIN {X 0,Y 425.31,Z 331.134,A -85,B 0,C 180,E1 -9771.102,E2 -9771.102} C_VEL
LIN {X 0,Y 425.302,Z 331.135,A -85,B 0,C 180,E1 -9774.664,E2 -9774.664} C_VEL
LIN {X 0,Y 425.266,Z 331.138,A -85,B 0,C 180,E1 -9778.073,E2 -9778.073} C_VEL
LIN {X 0,Y 425.333,Z 331.24,A -85,B 0,C 180,E1 -9780.61,E2 -9780.61} C_VEL
LIN {X 0,Y 428.185,Z 344.051,A -85,B 0,C 180,E1 -9783.168,E2 -9783.168} C_VEL
LIN {X 0,Y 429.346,Z 350.332,A -85,B 0,C 180,E1 -9784.379,E2 -9784.379} C_VEL
LIN {X 0,Y 428.224,Z 368.021,A -85,B 0,C 180,E1 -9787.505,E2 -9787.505} C_VEL
LIN {X 0,Y 433.048,Z 396.035,A -85,B 0,C 180,E1 -9788.236,E2 -9788.236} C_VEL
LIN {X 0,Y 431.617,Z 505.012,A -85,B 0,C 180,E1 -9790.067,E2 -9790.067} C_VEL
LIN {X 0,Y 431.089,Z 519.405,A -85,B 0,C 180,E1 -9790.475,E2 -9790.475} C_VEL
LIN {X 0,Y 430.446,Z 532.684,A -85,B 0,C 180,E1 -9791.035,E2 -9791.035} C_VEL
LIN {X 0,Y 429.683,Z 545.808,A -85,B 0,C 180,E1 -9791.778,E2 -9791.778} C_VEL
LIN {X 0,Y 428.764,Z 558.762,A -85,B 0,C 180,E1 -9792.717,E2 -9792.717} C_VEL
LIN {X 0,Y 427.819,Z 570.592,A -85,B 0,C 180,E1 -9793.783,E2 -9793.783} C_VEL
LIN {X 0,Y 426.969,Z 581.412,A -85,B 0,C 180,E1 -9794.974,E2 -9794.974} C_VEL
LIN {X 0,Y 426.225,Z 590.475,A -85,B 0,C 180,E1 -9796.167,E2 -9796.167} C_VEL
LIN {X 0,Y 425.607,Z 599.586,A -85,B 0,C 180,E1 -9797.604,E2 -9797.604} C_VEL
LIN {X 0,Y 425.069,Z 607.166,A -85,B 0,C 180,E1 -9799.039,E2 -9799.039} C_VEL
LIN {X 0,Y 424.676,Z 613.488,A -85,B 0,C 180,E1 -9800.474,E2 -9800.474} C_VEL
LIN {X 0,Y 424.335,Z 620.178,A -85,B 0,C 180,E1 -9802.386,E2 -9802.386} C_VEL
LIN {X 0,Y 424.252,Z 623.797,A -85,B 0,C 180,E1 -9803.688,E2 -9803.688} C_VEL
LIN {X 0,Y 424.171,Z 627.136,A -85,B 0,C 180,E1 -9805.248,E2 -9805.248} C_VEL
LIN {X 0,Y 424.128,Z 629.932,A -85,B 0,C 180,E1 -9807.151,E2 -9807.151} C_VEL
LIN {X 0,Y 424.086,Z 631.355,A -85,B 0,C 180,E1 -9809.05,E2 -9809.05} C_VEL
LIN {X 0,Y 424.086,Z 631.439,A -85,B 0,C 180,E1 -9810.95,E2 -9810.95} C_VEL
LIN {X 0,Y 424.126,Z 630.19,A -85,B 0,C 180,E1 -9812.849,E2 -9812.849} C_VEL
LIN {X 0,Y 424.171,Z 627.574,A -85,B 0,C 180,E1 -9814.752,E2 -9814.752} C_VEL
LIN {X 0,Y 424.294,Z 623.514,A -85,B 0,C 180,E1 -9816.658,E2 -9816.658} C_VEL
LIN {X 0,Y 424.5,Z 617.905,A -85,B 0,C 180,E1 -9818.569,E2 -9818.569} C_VEL
LIN {X 0,Y 424.87,Z 611.59,A -85,B 0,C 180,E1 -9820.243,E2 -9820.243} C_VEL
LIN {X 0,Y 425.556,Z 603.745,A -85,B 0,C 180,E1 -9821.914,E2 -9821.914} C_VEL
LIN {X 0,Y 426.121,Z 595.562,A -85,B 0,C 180,E1 -9823.35,E2 -9823.35} C_VEL
LIN {X 0,Y 426.982,Z 585.723,A -85,B 0,C 180,E1 -9824.781,E2 -9824.781} C_VEL
LIN {X 0,Y 427.926,Z 574.809,A -85,B 0,C 180,E1 -9826.09,E2 -9826.09} C_VEL
LIN {X 0,Y 429.118,Z 562.715,A -85,B 0,C 180,E1 -9827.268,E2 -9827.268} C_VEL
LIN {X 0,Y 430.048,Z 550.613,A -85,B 0,C 180,E1 -9828.225,E2 -9828.225} C_VEL
LIN {X 0,Y 430.992,Z 536.504,A -85,B 0,C 180,E1 -9829.096,E2 -9829.096} C_VEL
LIN {X 0,Y 431.71,Z 523.273,A -85,B 0,C 180,E1 -9829.712,E2 -9829.712} C_VEL
LIN {X 0,Y 432.39,Z 508.909,A -85,B 0,C 180,E1 -9830.175,E2 -9830.175} C_VEL
LIN {X 0,Y 432.786,Z 488.928,A -85,B 0,C 180,E1 -9830.559,E2 -9830.559} C_VEL
LIN {X 0,Y 434.076,Z 395.878,A -85,B 0,C 180,E1 -9832.127,E2 -9832.127} C_VEL
LIN {X 0,Y 429.872,Z 373.42,A -85,B 0,C 180,E1 -9832.774,E2 -9832.774} C_VEL
LIN {X 0,Y 428.699,Z 367.812,A -85,B 0,C 180,E1 -9832.964,E2 -9832.964} C_VEL
LIN {X 0,Y 429.981,Z 352.273,A -85,B 0,C 180,E1 -9835.756,E2 -9835.756} C_VEL
LIN {X 0,Y 427.818,Z 341.474,A -85,B 0,C 180,E1 -9837.94,E2 -9837.94} C_VEL
LIN {X 0,Y 425.316,Z 331.128,A -85,B 0,C 180,E1 -9840.162,E2 -9840.162} C_VEL
LIN {X 0,Y 425.284,Z 331.134,A -85,B 0,C 180,E1 -9843.048,E2 -9843.048} C_VEL
LIN {X 0,Y 425.284,Z 331.135,A -85,B 0,C 180,E1 -9845.929,E2 -9845.929} C_VEL
LIN {X 0,Y 425.289,Z 331.13,A -85,B 0,C 180,E1 -9849.042,E2 -9849.042} C_VEL
LIN {X 0,Y 425.291,Z 331.132,A -85,B 0,C 180,E1 -9851.958,E2 -9851.958} C_VEL
LIN {X 0,Y 425.286,Z 331.13,A -85,B 0,C 180,E1 -9855.283,E2 -9855.283} C_VEL
LIN {X 0,Y 425.277,Z 331.136,A -85,B 0,C 180,E1 -9858.622,E2 -9858.622} C_VEL
LIN {X 0,Y 425.314,Z 331.127,A -85,B 0,C 180,E1 -9861.103,E2 -9861.103} C_VEL
LIN {X 0,Y 425.301,Z 331.133,A -85,B 0,C 180,E1 -9864.664,E2 -9864.664} C_VEL
LIN {X 0,Y 425.268,Z 331.137,A -85,B 0,C 180,E1 -9868.073,E2 -9868.073} C_VEL
LIN {X 0,Y 425.316,Z 331.127,A -85,B 0,C 180,E1 -9871.367,E2 -9871.367} C_VEL
LIN {X 0,Y 425.276,Z 331.136,A -85,B 0,C 180,E1 -9874.554,E2 -9874.554} C_VEL
LIN {X 0,Y 425.288,Z 331.131,A -85,B 0,C 180,E1 -9876.634,E2 -9876.634} C_VEL
LIN {X 0,Y 425.299,Z 331.131,A -85,B 0,C 180,E1 -9879.695,E2 -9879.695} C_VEL
LIN {X 0,Y 425.342,Z 331.123,A -85,B 0,C 180,E1 -9882.698,E2 -9882.698} C_VEL
LIN {X 0,Y 425.351,Z 331.126,A -85,B 0,C 180,E1 -9885.65,E2 -9885.65} C_VEL
LIN {X 0,Y 425.353,Z 331.125,A -85,B 0,C 180,E1 -9888.564,E2 -9888.564} C_VEL
LIN {X 0,Y 425.411,Z 331.114,A -85,B 0,C 180,E1 -9891.45,E2 -9891.45} C_VEL
LIN {X 0,Y 425.535,Z 331.103,A -85,B 0,C 180,E1 -9894.313,E2 -9894.313} C_VEL
LIN {X 0,Y 425.569,Z 331.1,A -85,B 0,C 180,E1 -9898.108,E2 -9898.108} C_VEL
LIN {X 0,Y 425.594,Z 331.096,A -85,B 0,C 180,E1 -9900,E2 -9900} C_VEL
LIN {X 0,Y 425.538,Z 331.097,A -85,B 0,C 180,E1 -9902.84,E2 -9902.84} C_VEL
LIN {X 0,Y 425.48,Z 331.1,A -85,B 0,C 180,E1 -9906.483,E2 -9906.483} C_VEL
LIN {X 0,Y 425.399,Z 331.121,A -85,B 0,C 180,E1 -9909.51,E2 -9909.51} C_VEL
LIN {X 0,Y 425.398,Z 331.115,A -85,B 0,C 180,E1 -9912.904,E2 -9912.904} C_VEL
LIN {X 0,Y 425.317,Z 331.122,A -85,B 0,C 180,E1 -9916.583,E2 -9916.583} C_VEL
LIN {X 0,Y 425.3,Z 331.132,A -85,B 0,C 180,E1 -9919.623,E2 -9919.623} C_VEL
LIN {X 0,Y 425.29,Z 331.132,A -85,B 0,C 180,E1 -9922.339,E2 -9922.339} C_VEL
LIN {X 0,Y 425.263,Z 331.134,A -85,B 0,C 180,E1 -9925.448,E2 -9925.448} C_VEL
LIN {X 0,Y 425.299,Z 331.126,A -85,B 0,C 180,E1 -9928.857,E2 -9928.857} C_VEL
LIN {X 0,Y 425.256,Z 331.134,A -85,B 0,C 180,E1 -9931.928,E2 -9931.928} C_VEL
LIN {X 0,Y 425.295,Z 331.126,A -85,B 0,C 180,E1 -9935.337,E2 -9935.337} C_VEL
LIN {X 0,Y 425.268,Z 331.135,A -85,B 0,C 180,E1 -9938.903,E2 -9938.903} C_VEL
LIN {X 0,Y 425.265,Z 331.135,A -85,B 0,C 180,E1 -9941.954,E2 -9941.954} C_VEL
LIN {X 0,Y 425.286,Z 331.13,A -85,B 0,C 180,E1 -9945.284,E2 -9945.284} C_VEL
LIN {X 0,Y 425.248,Z 331.14,A -85,B 0,C 180,E1 -9948.618,E2 -9948.618} C_VEL
LIN {X 0,Y 425.27,Z 331.138,A -85,B 0,C 180,E1 -9952.304,E2 -9952.304} C_VEL
LIN {X 0,Y 425.286,Z 331.134,A -85,B 0,C 180,E1 -9955.815,E2 -9955.815} C_VEL
LIN {X 0,Y 425.297,Z 331.176,A -85,B 0,C 180,E1 -9958.563,E2 -9958.563} C_VEL
LIN {X 0,Y 428.073,Z 344.086,A -85,B 0,C 180,E1 -9961.568,E2 -9961.568} C_VEL
LIN {X 0,Y 428.538,Z 346.405,A -85,B 0,C 180,E1 -9962.092,E2 -9962.092} C_VEL
LIN {X 0,Y 430.897,Z 353.739,A -85,B 0,C 180,E1 -9962.374,E2 -9962.374} C_VEL
LIN {X 0,Y 434.376,Z 369.251,A -85,B 0,C 180,E1 -9962.859,E2 -9962.859} C_VEL
LIN {X 0,Y 432.829,Z 482.984,A -85,B 0,C 180,E1 -9964.803,E2 -9964.803} C_VEL
LIN {X 0,Y 432.299,Z 497.548,A -85,B 0,C 180,E1 -9965.242,E2 -9965.242} C_VEL
LIN {X 0,Y 431.472,Z 511.499,A -85,B 0,C 180,E1 -9965.855,E2 -9965.855} C_VEL
LIN {X 0,Y 430.669,Z 525.359,A -85,B 0,C 180,E1 -9966.688,E2 -9966.688} C_VEL
LIN {X 0,Y 429.698,Z 537.902,A -85,B 0,C 180,E1 -9967.649,E2 -9967.649} C_VEL
LIN {X 0,Y 428.759,Z 549.329,A -85,B 0,C 180,E1 -9968.736,E2 -9968.736} C_VEL
LIN {X 0,Y 427.752,Z 560.769,A -85,B 0,C 180,E1 -9970.067,E2 -9970.067} C_VEL
LIN {X 0,Y 426.804,Z 570.93,A -85,B 0,C 180,E1 -9971.519,E2 -9971.519} C_VEL
LIN {X 0,Y 426.463,Z 574.652,A -85,B 0,C 180,E1 -9972.13,E2 -9972.13} C_VEL
LIN {X 0,Y 425.51,Z 578.289,A -85,B 0,C 180,E1 -9972.749,E2 -9972.749} C_VEL
LIN {X 0,Y 422.172,Z 583.867,A -85,B 0,C 180,E1 -9973.762,E2 -9973.762} C_VEL
LIN {X 0,Y 418.877,Z 588.949,A -85,B 0,C 180,E1 -9974.834,E2 -9974.834} C_VEL
LIN {X 0,Y 418.003,Z 591.69,A -85,B 0,C 180,E1 -9975.539,E2 -9975.539} C_VEL
LIN {X 0,Y 417.541,Z 597.53,A -85,B 0,C 180,E1 -9977.36,E2 -9977.36} C_VEL
LIN {X 0,Y 417.25,Z 602.239,A -85,B 0,C 180,E1 -9979.322,E2 -9979.322} C_VEL
LIN {X 0,Y 417.074,Z 605.417,A -85,B 0,C 180,E1 -9981.277,E2 -9981.277} C_VEL
LIN {X 0,Y 417.033,Z 607.205,A -85,B 0,C 180,E1 -9983.225,E2 -9983.225} C_VEL
LIN {X 0,Y 417.035,Z 607.665,A -85,B 0,C 180,E1 -9985.166,E2 -9985.166} C_VEL
LIN {X 0,Y 417.059,Z 606.808,A -85,B 0,C 180,E1 -9987.102,E2 -9987.102} C_VEL
LIN {X 0,Y 417.041,Z 604.63,A -85,B 0,C 180,E1 -9989.034,E2 -9989.034} C_VEL
LIN {X 0,Y 417.161,Z 601.074,A -85,B 0,C 180,E1 -9990.965,E2 -9990.965} C_VEL
LIN {X 0,Y 417.464,Z 596.037,A -85,B 0,C 180,E1 -9992.895,E2 -9992.895} C_VEL
LIN {X 0,Y 417.969,Z 591.151,A -85,B 0,C 180,E1 -9994.339,E2 -9994.339} C_VEL
LIN {X 0,Y 418.53,Z 584.156,A -85,B 0,C 180,E1 -9996.024,E2 -9996.024} C_VEL
LIN {X 0,Y 419.149,Z 575.521,A -85,B 0,C 180,E1 -9997.709,E2 -9997.709} C_VEL
LIN {X 0,Y 419.682,Z 568.101,A -85,B 0,C 180,E1 -9998.911,E2 -9998.911} C_VEL
LIN {X 0,Y 420.709,Z 557.481,A -85,B 0,C 180,E1 -10000.345,E2 -10000.345} C_VEL
LIN {X 0,Y 421.608,Z 545.599,A -85,B 0,C 180,E1 -10001.661,E2 -10001.661} C_VEL
LIN {X 0,Y 422.529,Z 533.605,A -85,B 0,C 180,E1 -10002.732,E2 -10002.732} C_VEL
LIN {X 0,Y 423.316,Z 522.083,A -85,B 0,C 180,E1 -10003.563,E2 -10003.563} C_VEL
LIN {X 0,Y 424.164,Z 508.463,A -85,B 0,C 180,E1 -10004.33,E2 -10004.33} C_VEL
LIN {X 0,Y 424.707,Z 494.978,A -85,B 0,C 180,E1 -10004.893,E2 -10004.893} C_VEL
LIN {X 0,Y 425.074,Z 481.349,A -85,B 0,C 180,E1 -10005.278,E2 -10005.278} C_VEL
LIN {X 0,Y 426.559,Z 369.499,A -85,B 0,C 180,E1 -10007.188,E2 -10007.188} C_VEL
LIN {X 0,Y 421.872,Z 348.504,A -85,B 0,C 180,E1 -10007.805,E2 -10007.805} C_VEL
LIN {X 0,Y 421.225,Z 346.37,A -85,B 0,C 180,E1 -10007.901,E2 -10007.901} C_VEL
LIN {X 0,Y 418.34,Z 332.45,A -85,B 0,C 180,E1 -10011.045,E2 -10011.045} C_VEL
LIN {X 0,Y 418.262,Z 332.013,A -85,B 0,C 180,E1 -10011.178,E2 -10011.178} C_VEL
LIN {X 0,Y 418.248,Z 332.016,A -85,B 0,C 180,E1 -10014.852,E2 -10014.852} C_VEL
LIN {X 0,Y 418.203,Z 332.017,A -85,B 0,C 180,E1 -10018.07,E2 -10018.07} C_VEL
LIN {X 0,Y 418.236,Z 332.013,A -85,B 0,C 180,E1 -10021.018,E2 -10021.018} C_VEL
LIN {X 0,Y 418.23,Z 332.011,A -85,B 0,C 180,E1 -10023.679,E2 -10023.679} C_VEL
LIN {X 0,Y 418.233,Z 332.013,A -85,B 0,C 180,E1 -10027.225,E2 -10027.225} C_VEL
LIN {X 0,Y 418.208,Z 332.016,A -85,B 0,C 180,E1 -10030.95,E2 -10030.95} C_VEL
LIN {X 0,Y 418.203,Z 332.014,A -85,B 0,C 180,E1 -10033.728,E2 -10033.728} C_VEL
LIN {X 0,Y 418.201,Z 332.017,A -85,B 0,C 180,E1 -10036.447,E2 -10036.447} C_VEL
LIN {X 0,Y 418.208,Z 332.013,A -85,B 0,C 180,E1 -10039.133,E2 -10039.133} C_VEL
LIN {X 0,Y 418.235,Z 332.01,A -85,B 0,C 180,E1 -10042.775,E2 -10042.775} C_VEL
LIN {X 0,Y 418.234,Z 332.013,A -85,B 0,C 180,E1 -10046.321,E2 -10046.321} C_VEL
LIN {X 0,Y 418.236,Z 332.01,A -85,B 0,C 180,E1 -10049.727,E2 -10049.727} C_VEL
LIN {X 0,Y 418.211,Z 332.01,A -85,B 0,C 180,E1 -10053.016,E2 -10053.016} C_VEL
LIN {X 0,Y 418.261,Z 332.012,A -85,B 0,C 180,E1 -10056.217,E2 -10056.217} C_VEL
LIN {X 0,Y 418.25,Z 331.991,A -85,B 0,C 180,E1 -10059.337,E2 -10059.337} C_VEL
LIN {X 0,Y 418.255,Z 332.008,A -85,B 0,C 180,E1 -10062.394,E2 -10062.394} C_VEL
LIN {X 0,Y 418.281,Z 332.003,A -85,B 0,C 180,E1 -10065.402,E2 -10065.402} C_VEL
LIN {X 0,Y 418.317,Z 331.983,A -85,B 0,C 180,E1 -10068.369,E2 -10068.369} C_VEL
LIN {X 0,Y 418.381,Z 331.985,A -85,B 0,C 180,E1 -10071.304,E2 -10071.304} C_VEL
LIN {X 0,Y 418.488,Z 331.983,A -85,B 0,C 180,E1 -10074.217,E2 -10074.217} C_VEL
LIN {X 0,Y 418.543,Z 331.976,A -85,B 0,C 180,E1 -10078.075,E2 -10078.075} C_VEL
LIN {X 0,Y 418.476,Z 331.975,A -85,B 0,C 180,E1 -10080.962,E2 -10080.962} C_VEL
LIN {X 0,Y 418.476,Z 331.98,A -85,B 0,C 180,E1 -10082.888,E2 -10082.888} C_VEL
LIN {X 0,Y 418.492,Z 331.978,A -85,B 0,C 180,E1 -10085.783,E2 -10085.783} C_VEL
LIN {X 0,Y 418.38,Z 331.991,A -85,B 0,C 180,E1 -10088.695,E2 -10088.695} C_VEL
LIN {X 0,Y 418.317,Z 332.001,A -85,B 0,C 180,E1 -10091.631,E2 -10091.631} C_VEL
LIN {X 0,Y 418.305,Z 331.999,A -85,B 0,C 180,E1 -10094.597,E2 -10094.597} C_VEL
LIN {X 0,Y 418.288,Z 332.007,A -85,B 0,C 180,E1 -10097.604,E2 -10097.604} C_VEL
LIN {X 0,Y 418.253,Z 332.007,A -85,B 0,C 180,E1 -10100.663,E2 -10100.663} C_VEL
LIN {X 0,Y 418.288,Z 332.009,A -85,B 0,C 180,E1 -10103.781,E2 -10103.781} C_VEL
LIN {X 0,Y 418.268,Z 332.007,A -85,B 0,C 180,E1 -10107.058,E2 -10107.058} C_VEL
LIN {X 0,Y 418.246,Z 332.012,A -85,B 0,C 180,E1 -10110.272,E2 -10110.272} C_VEL
LIN {X 0,Y 418.251,Z 332.015,A -85,B 0,C 180,E1 -10113.677,E2 -10113.677} C_VEL
LIN {X 0,Y 418.247,Z 332.013,A -85,B 0,C 180,E1 -10117.223,E2 -10117.223} C_VEL
LIN {X 0,Y 418.257,Z 332.015,A -85,B 0,C 180,E1 -10119.681,E2 -10119.681} C_VEL
LIN {X 0,Y 418.231,Z 332.012,A -85,B 0,C 180,E1 -10122.321,E2 -10122.321} C_VEL
LIN {X 0,Y 418.237,Z 332.013,A -85,B 0,C 180,E1 -10125.108,E2 -10125.108} C_VEL
LIN {X 0,Y 418.241,Z 332.012,A -85,B 0,C 180,E1 -10127.767,E2 -10127.767} C_VEL
LIN {X 0,Y 418.258,Z 332.014,A -85,B 0,C 180,E1 -10131.559,E2 -10131.559} C_VEL
LIN {X 0,Y 418.261,Z 332.015,A -85,B 0,C 180,E1 -10135.159,E2 -10135.159} C_VEL
LIN {X 0,Y 418.247,Z 332.016,A -85,B 0,C 180,E1 -10137.472,E2 -10137.472} C_VEL
LIN {X 0,Y 418.299,Z 332.205,A -85,B 0,C 180,E1 -10140.326,E2 -10140.326} C_VEL
LIN {X 0,Y 421.23,Z 345.303,A -85,B 0,C 180,E1 -10142.994,E2 -10142.994} C_VEL
LIN {X 0,Y 422.43,Z 352.348,A -85,B 0,C 180,E1 -10144.369,E2 -10144.369} C_VEL
LIN {X 0,Y 421.372,Z 367.817,A -85,B 0,C 180,E1 -10147.149,E2 -10147.149} C_VEL
LIN {X 0,Y 426.392,Z 397.618,A -85,B 0,C 180,E1 -10147.939,E2 -10147.939} C_VEL
LIN {X 0,Y 424.875,Z 504.962,A -85,B 0,C 180,E1 -10149.768,E2 -10149.768} C_VEL
LIN {X 0,Y 424.352,Z 519.288,A -85,B 0,C 180,E1 -10150.184,E2 -10150.184} C_VEL
LIN {X 0,Y 423.624,Z 533.432,A -85,B 0,C 180,E1 -10150.798,E2 -10150.798} C_VEL
LIN {X 0,Y 422.783,Z 546.896,A -85,B 0,C 180,E1 -10151.588,E2 -10151.588} C_VEL
LIN {X 0,Y 421.821,Z 559.68,A -85,B 0,C 180,E1 -10152.548,E2 -10152.548} C_VEL
LIN {X 0,Y 420.854,Z 571.314,A -85,B 0,C 180,E1 -10153.632,E2 -10153.632} C_VEL
LIN {X 0,Y 419.885,Z 582.962,A -85,B 0,C 180,E1 -10154.963,E2 -10154.963} C_VEL
LIN {X 0,Y 419.158,Z 591.738,A -85,B 0,C 180,E1 -10156.177,E2 -10156.177} C_VEL
LIN {X 0,Y 418.493,Z 600.604,A -85,B 0,C 180,E1 -10157.636,E2 -10157.636} C_VEL
LIN {X 0,Y 417.953,Z 607.971,A -85,B 0,C 180,E1 -10159.095,E2 -10159.095} C_VEL
LIN {X 0,Y 417.511,Z 615.018,A -85,B 0,C 180,E1 -10160.798,E2 -10160.798} C_VEL
LIN {X 0,Y 417.246,Z 621.341,A -85,B 0,C 180,E1 -10162.743,E2 -10162.743} C_VEL
LIN {X 0,Y 417.111,Z 624.943,A -85,B 0,C 180,E1 -10164.198,E2 -10164.198} C_VEL
LIN {X 0,Y 417.003,Z 628.469,A -85,B 0,C 180,E1 -10166.135,E2 -10166.135} C_VEL
LIN {X 0,Y 417.053,Z 630.592,A -85,B 0,C 180,E1 -10168.069,E2 -10168.069} C_VEL
LIN {X 0,Y 417.002,Z 631.359,A -85,B 0,C 180,E1 -10170,E2 -10170} C_VEL
LIN {X 0,Y 417.053,Z 630.795,A -85,B 0,C 180,E1 -10171.931,E2 -10171.931} C_VEL
LIN {X 0,Y 417.002,Z 628.887,A -85,B 0,C 180,E1 -10173.866,E2 -10173.866} C_VEL
LIN {X 0,Y 417.111,Z 625.582,A -85,B 0,C 180,E1 -10175.802,E2 -10175.802} C_VEL
LIN {X 0,Y 417.242,Z 622.125,A -85,B 0,C 180,E1 -10177.258,E2 -10177.258} C_VEL
LIN {X 0,Y 417.537,Z 616.164,A -85,B 0,C 180,E1 -10179.201,E2 -10179.201} C_VEL
LIN {X 0,Y 417.999,Z 609.463,A -85,B 0,C 180,E1 -10180.903,E2 -10180.903} C_VEL
LIN {X 0,Y 418.701,Z 601.138,A -85,B 0,C 180,E1 -10182.604,E2 -10182.604} C_VEL
LIN {X 0,Y 419.459,Z 592.478,A -85,B 0,C 180,E1 -10184.061,E2 -10184.061} C_VEL
LIN {X 0,Y 420.411,Z 582.002,A -85,B 0,C 180,E1 -10185.514,E2 -10185.514} C_VEL
LIN {X 0,Y 421.549,Z 570.298,A -85,B 0,C 180,E1 -10186.839,E2 -10186.839} C_VEL
LIN {X 0,Y 422.619,Z 558.594,A -85,B 0,C 180,E1 -10187.918,E2 -10187.918} C_VEL
LIN {X 0,Y 423.63,Z 546.21,A -85,B 0,C 180,E1 -10188.84,E2 -10188.84} C_VEL
LIN {X 0,Y 424.569,Z 532.308,A -85,B 0,C 180,E1 -10189.648,E2 -10189.648} C_VEL
LIN {X 0,Y 425.372,Z 518.39,A -85,B 0,C 180,E1 -10190.239,E2 -10190.239} C_VEL
LIN {X 0,Y 425.974,Z 503.653,A -85,B 0,C 180,E1 -10190.65,E2 -10190.65} C_VEL
LIN {X 0,Y 427.59,Z 397.759,A -85,B 0,C 180,E1 -10192.472,E2 -10192.472} C_VEL
LIN {X 0,Y 425.078,Z 382.77,A -85,B 0,C 180,E1 -10192.895,E2 -10192.895} C_VEL
LIN {X 0,Y 421.943,Z 367.53,A -85,B 0,C 180,E1 -10193.399,E2 -10193.399} C_VEL
LIN {X 0,Y 423.079,Z 353.397,A -85,B 0,C 180,E1 -10195.991,E2 -10195.991} C_VEL
LIN {X 0,Y 420.932,Z 342.98,A -85,B 0,C 180,E1 -10198.143,E2 -10198.143} C_VEL
LIN {X 0,Y 418.253,Z 332.004,A -85,B 0,C 180,E1 -10200.545,E2 -10200.545} C_VEL
LIN {X 0,Y 418.25,Z 332.008,A -85,B 0,C 180,E1 -10203.677,E2 -10203.677} C_VEL
LIN {X 0,Y 418.241,Z 332.012,A -85,B 0,C 180,E1 -10207.224,E2 -10207.224} C_VEL
LIN {X 0,Y 418.248,Z 332.008,A -85,B 0,C 180,E1 -10209.683,E2 -10209.683} C_VEL
LIN {X 0,Y 418.231,Z 332.015,A -85,B 0,C 180,E1 -10212.321,E2 -10212.321} C_VEL
LIN {X 0,Y 418.237,Z 332.009,A -85,B 0,C 180,E1 -10215.109,E2 -10215.109} C_VEL
LIN {X 0,Y 418.242,Z 332.009,A -85,B 0,C 180,E1 -10217.767,E2 -10217.767} C_VEL
LIN {X 0,Y 418.26,Z 332.007,A -85,B 0,C 180,E1 -10220.619,E2 -10220.619} C_VEL
LIN {X 0,Y 418.244,Z 332.008,A -85,B 0,C 180,E1 -10223.976,E2 -10223.976} C_VEL
LIN {X 0,Y 418.26,Z 332.005,A -85,B 0,C 180,E1 -10227.156,E2 -10227.156} C_VEL
LIN {X 0,Y 418.263,Z 332.007,A -85,B 0,C 180,E1 -10230.838,E2 -10230.838} C_VEL
LIN {X 0,Y 418.24,Z 332.009,A -85,B 0,C 180,E1 -10234.094,E2 -10234.094} C_VEL
LIN {X 0,Y 418.235,Z 332.007,A -85,B 0,C 180,E1 -10237.264,E2 -10237.264} C_VEL
LIN {X 0,Y 418.286,Z 332.006,A -85,B 0,C 180,E1 -10240.365,E2 -10240.365} C_VEL
LIN {X 0,Y 418.32,Z 331.997,A -85,B 0,C 180,E1 -10243.405,E2 -10243.405} C_VEL
LIN {X 0,Y 418.35,Z 331.989,A -85,B 0,C 180,E1 -10247,E2 -10247} C_VEL
LIN {X 0,Y 418.341,Z 331.996,A -85,B 0,C 180,E1 -10250.329,E2 -10250.329} C_VEL
LIN {X 0,Y 418.447,Z 331.982,A -85,B 0,C 180,E1 -10253.248,E2 -10253.248} C_VEL
LIN {X 0,Y 418.326,Z 331.998,A -85,B 0,C 180,E1 -10255.182,E2 -10255.182} C_VEL
LIN {X 0,Y 418.538,Z 331.975,A -85,B 0,C 180,E1 -10258.076,E2 -10258.076} C_VEL
LIN {X 0,Y 418.547,Z 331.974,A -85,B 0,C 180,E1 -10260,E2 -10260} C_VEL
LIN {X 0,Y 418.493,Z 331.975,A -85,B 0,C 180,E1 -10262.888,E2 -10262.888} C_VEL
LIN {X 0,Y 418.444,Z 331.976,A -85,B 0,C 180,E1 -10266.481,E2 -10266.481} C_VEL
LIN {X 0,Y 418.38,Z 331.992,A -85,B 0,C 180,E1 -10268.696,E2 -10268.696} C_VEL
LIN {X 0,Y 418.318,Z 331.998,A -85,B 0,C 180,E1 -10271.631,E2 -10271.631} C_VEL
LIN {X 0,Y 418.281,Z 332.004,A -85,B 0,C 180,E1 -10274.598,E2 -10274.598} C_VEL
LIN {X 0,Y 418.241,Z 332.01,A -85,B 0,C 180,E1 -10277.606,E2 -10277.606} C_VEL
LIN {X 0,Y 418.24,Z 332.004,A -85,B 0,C 180,E1 -10280.664,E2 -10280.664} C_VEL
LIN {X 0,Y 418.259,Z 332.008,A -85,B 0,C 180,E1 -10283.783,E2 -10283.783} C_VEL
LIN {X 0,Y 418.209,Z 332.015,A -85,B 0,C 180,E1 -10287.042,E2 -10287.042} C_VEL
LIN {X 0,Y 418.237,Z 331.991,A -85,B 0,C 180,E1 -10290.273,E2 -10290.273} C_VEL
LIN {X 0,Y 418.235,Z 332.014,A -85,B 0,C 180,E1 -10293.679,E2 -10293.679} C_VEL
LIN {X 0,Y 418.235,Z 332,A -85,B 0,C 180,E1 -10297.225,E2 -10297.225} C_VEL
LIN {X 0,Y 418.208,Z 332.014,A -85,B 0,C 180,E1 -10300.95,E2 -10300.95} C_VEL
LIN {X 0,Y 418.204,Z 332.018,A -85,B 0,C 180,E1 -10303.728,E2 -10303.728} C_VEL
LIN {X 0,Y 418.201,Z 332.012,A -85,B 0,C 180,E1 -10306.447,E2 -10306.447} C_VEL
LIN {X 0,Y 418.208,Z 332.014,A -85,B 0,C 180,E1 -10309.133,E2 -10309.133} C_VEL
LIN {X 0,Y 418.234,Z 332.016,A -85,B 0,C 180,E1 -10312.775,E2 -10312.775} C_VEL
LIN {X 0,Y 418.23,Z 332.012,A -85,B 0,C 180,E1 -10316.321,E2 -10316.321} C_VEL
LIN {X 0,Y 418.239,Z 332.157,A -85,B 0,C 180,E1 -10318.217,E2 -10318.217} C_VEL
LIN {X 0,Y 420.878,Z 343.972,A -85,B 0,C 180,E1 -10321.036,E2 -10321.036} C_VEL
LIN {X 0,Y 421.431,Z 346.766,A -85,B 0,C 180,E1 -10321.656,E2 -10321.656} C_VEL
